	{attribute 'TcIecLibraryType'}
	{attribute 'external_name' := 'F_VN_DrawArrow_GUID_A67F059E_E66C_28C8_6DC9_666EC4C23162'}
	(* Draw an arrowed line. *)
	FUNCTION F_VN_DrawArrow : HRESULT
	VAR_INPUT
		nX1	:	UDINT;	(* x coordinate of the start point *)
		nY1	:	UDINT;	(* y coordinate of the start point *)
		nX2	:	UDINT;	(* x coordinate of the end point *)
		nY2	:	UDINT;	(* y coordinate of the end point *)
		ipDestImage	:	ITcVnImage;	(* Destination image *)
	END_VAR
	VAR_IN_OUT
		aColor	:	TcVnVector4_LREAL;	(* Color *)
	END_VAR
	VAR_INPUT
		nThickness	:	DINT;	(* Line thickness *)
		bDoubleHead	:	BOOL;	(* To draw an arrow on each side of the line. *)
		hrPrev	:	HRESULT;	(* HRESULT indicating the result of previous operations (If SUCCEEDED(hrPrev) equals false, no operation is executed.) *)
	END_VAR

END_FUNCTION

// Functions/Drawing/F_VN_DrawArrow_TcVnVector4_DINT

	{attribute 'TcIecLibraryType'}
	{attribute 'external_name' := 'F_VN_DrawArrow_TcVnVector4_DINT_GUID_4A77EF94_9C2A_22D4_5693_A510294A7600'}
	(* Draw an arrowed line. *)
	FUNCTION F_VN_DrawArrow_TcVnVector4_DINT : HRESULT
	VAR_IN_OUT
		aLine	:	TcVnVector4_DINT;	(* The start and end point of a line segment [x1, y1, x2, y2] *)
	END_VAR
	VAR_INPUT
		ipDestImage	:	ITcVnImage;	(* Destination image *)
	END_VAR
	VAR_IN_OUT
		aColor	:	TcVnVector4_LREAL;	(* Color *)
	END_VAR
	VAR_INPUT
		nThickness	:	DINT;	(* Line thickness *)
		bDoubleHead	:	BOOL;	(* To draw an arrow on each side of the line. *)
		hrPrev	:	HRESULT;	(* HRESULT indicating the result of previous operations (If SUCCEEDED(hrPrev) equals false, no operation is executed.) *)
	END_VAR

END_FUNCTION

// Functions/Drawing/F_VN_DrawArrowExp

	{attribute 'TcIecLibraryType'}
	{attribute 'external_name' := 'F_VN_DrawArrowExp_GUID_1F944010_3B82_22C2_4B5D_AA48D2E539AF'}
	(* Draws an arrowed line. (expert function) *)
	FUNCTION F_VN_DrawArrowExp : HRESULT
	VAR_INPUT
		nX1	:	UDINT;	(* x coordinate of the start point *)
		nY1	:	UDINT;	(* y coordinate of the start point *)
		nX2	:	UDINT;	(* x coordinate of the end point *)
		nY2	:	UDINT;	(* y coordinate of the end point *)
		ipDestImage	:	ITcVnImage;	(* Destination image *)
	END_VAR
	VAR_IN_OUT
		aColor	:	TcVnVector4_LREAL;	(* Color *)
	END_VAR
	VAR_INPUT
		nThickness	:	DINT;	(* Line thickness *)
		bDoubleHead	:	BOOL;	(* To draw an arrow on each side of the line. *)
		eLineType	:	ETcVnLineType;	(* Line type *)
		nShift	:	UDINT;	(* Fractional bits of the coordinates (bit shift) *)
		fTipLenght	:	LREAL;	(* Lenght of the arrow's tip as a fraction of the line's lenght *)
		hrPrev	:	HRESULT;	(* HRESULT indicating the result of previous operations (If SUCCEEDED(hrPrev) equals false, no operation is executed.) *)
	END_VAR

END_FUNCTION

// Functions/Drawing/F_VN_DrawArrowExp_TcVnVector4_DINT

	{attribute 'TcIecLibraryType'}
	{attribute 'external_name' := 'F_VN_DrawArrowExp_TcVnVector4_DINT_GUID_6CFFFCA4_FF10_2C86_53F7_A52292798831'}
	(* Draws an arrowed line. (expert function) *)
	FUNCTION F_VN_DrawArrowExp_TcVnVector4_DINT : HRESULT
	VAR_IN_OUT
		aLine	:	TcVnVector4_DINT;	(* The start and end point of a line segment [x1, y1, x2, y2] *)
	END_VAR
	VAR_INPUT
		ipDestImage	:	ITcVnImage;	(* Destination image *)
	END_VAR
	VAR_IN_OUT
		aColor	:	TcVnVector4_LREAL;	(* Color *)
	END_VAR
	VAR_INPUT
		nThickness	:	DINT;	(* Line thickness *)
		bDoubleHead	:	BOOL;	(* To draw an arrow on each side of the line. *)
		eLineType	:	ETcVnLineType;	(* Line type *)
		nShift	:	UDINT;	(* Fractional bits of the coordinates (bit shift) *)
		fTipLenght	:	LREAL;	(* Lenght of the arrow's tip as a fraction of the line's lenght *)
		hrPrev	:	HRESULT;	(* HRESULT indicating the result of previous operations (If SUCCEEDED(hrPrev) equals false, no operation is executed.) *)
	END_VAR

END_FUNCTION

// Functions/Drawing/F_VN_DrawCircle

	{attribute 'TcIecLibraryType'}
	{attribute 'external_name' := 'F_VN_DrawCircle_GUID_62AE57B7_83F4_253D_652A_20281E468BE3'}
	(* Draws a circle. *)
	FUNCTION F_VN_DrawCircle : HRESULT
	VAR_INPUT
		nCenterX	:	UDINT;	(* x coordinate of the center *)
		nCenterY	:	UDINT;	(* y coordinate of the center *)
		nRadius	:	UDINT;	(* Radius *)
		ipDestImage	:	ITcVnImage;	(* Destination image *)
	END_VAR
	VAR_IN_OUT
		aColor	:	TcVnVector4_LREAL;	(* Color *)
	END_VAR
	VAR_INPUT
		nThickness	:	DINT;	(* Line thickness (if negative, the circle is filled) *)
		hrPrev	:	HRESULT;	(* HRESULT indicating the result of previous operations (If SUCCEEDED(hrPrev) equals false, no operation is executed.) *)
	END_VAR

END_FUNCTION

// Functions/Drawing/F_VN_DrawCircleExp

	{attribute 'TcIecLibraryType'}
	{attribute 'external_name' := 'F_VN_DrawCircleExp_GUID_6C116C34_AD29_2F99_4F7E_E03E108A0E54'}
	(* Draws a circle. *)
	FUNCTION F_VN_DrawCircleExp : HRESULT
	VAR_INPUT
		nCenterX	:	UDINT;	(* x coordinate of the center *)
		nCenterY	:	UDINT;	(* y coordinate of the center *)
		nRadius	:	UDINT;	(* Radius *)
		ipDestImage	:	ITcVnImage;	(* Destination image *)
	END_VAR
	VAR_IN_OUT
		aColor	:	TcVnVector4_LREAL;	(* Color *)
	END_VAR
	VAR_INPUT
		nThickness	:	DINT;	(* Line thickness (if negative, the circle is filled) *)
		eLineType	:	ETcVnLineType;	(* Line type *)
		hrPrev	:	HRESULT;	(* HRESULT indicating the result of previous operations (If SUCCEEDED(hrPrev) equals false, no operation is executed.) *)
	END_VAR

END_FUNCTION

// Functions/Drawing/F_VN_DrawCircles

	{attribute 'TcIecLibraryType'}
	{attribute 'external_name' := 'F_VN_DrawCircles_GUID_940A5C9B_16C1_20B9_6145_00E73CD7E7FA'}
	(* Draws circles. *)
	FUNCTION F_VN_DrawCircles : HRESULT
	VAR_INPUT
		ipCircles	:	ITcVnContainer;	(* Container with circles (ContainerType_Vector_TcVnVector3_REAL; Each container element contains the x coordinate of the circle center [0], the y coordinate of the circle center [1], and the radius [2].) *)
		nCircleIndex	:	DINT;	(* Index of a specific circle to be drawn (if negative, all circles within the container are drawn) *)
		ipDestImage	:	ITcVnImage;	(* Destination image *)
	END_VAR
	VAR_IN_OUT
		aColor	:	TcVnVector4_LREAL;	(* Color *)
	END_VAR
	VAR_INPUT
		nThickness	:	DINT;	(* Line thickness (if negative, the circle is filled) *)
		hrPrev	:	HRESULT;	(* HRESULT indicating the result of previous operations (If SUCCEEDED(hrPrev) equals false, no operation is executed.) *)
	END_VAR

END_FUNCTION

// Functions/Drawing/F_VN_DrawCirclesExp

	{attribute 'TcIecLibraryType'}
	{attribute 'external_name' := 'F_VN_DrawCirclesExp_GUID_C7646B92_088A_23BA_64E0_D477B3D449EC'}
	(* Draws circles. (expert function) *)
	FUNCTION F_VN_DrawCirclesExp : HRESULT
	VAR_INPUT
		ipCircles	:	ITcVnContainer;	(* Container with circles (ContainerType_Vector_TcVnVector3_REAL; Each container element contains the x coordinate of the circle center [0], the y coordinate of the circle center [1], and the radius [2].) *)
		nCircleIndex	:	DINT;	(* Index of a specific circle to be drawn (if negative, all circles within the container are drawn) *)
		ipDestImage	:	ITcVnImage;	(* Destination image *)
	END_VAR
	VAR_IN_OUT
		aColor	:	TcVnVector4_LREAL;	(* Color *)
	END_VAR
	VAR_INPUT
		nThickness	:	DINT;	(* Line thickness (if negative, the circle is filled) *)
		eLineType	:	ETcVnLineType;	(* Line type *)
		hrPrev	:	HRESULT;	(* HRESULT indicating the result of previous operations (If SUCCEEDED(hrPrev) equals false, no operation is executed.) *)
	END_VAR

END_FUNCTION

// Functions/Drawing/F_VN_DrawCircularArc

	{attribute 'TcIecLibraryType'}
	{attribute 'external_name' := 'F_VN_DrawCircularArc_GUID_65BA9826_3505_21EA_7421_EA736909BE51'}
	(* Draws a circular arc. *)
	FUNCTION F_VN_DrawCircularArc : HRESULT
	VAR_IN_OUT
		stCircularArc	:	TcVnCircularArc;	(* Circular arc definition *)
	END_VAR
	VAR_INPUT
		ipDestImage	:	ITcVnImage;	(* Destination image *)
	END_VAR
	VAR_IN_OUT
		aColor	:	TcVnVector4_LREAL;	(* Color *)
	END_VAR
	VAR_INPUT
		nThickness	:	DINT;	(* Line thickness (if negative, the arc is filled) *)
		hrPrev	:	HRESULT;	(* HRESULT indicating the result of previous operations (If SUCCEEDED(hrPrev) equals false, no operation is executed.) *)
	END_VAR

END_FUNCTION

// Functions/Drawing/F_VN_DrawCircularArcExp

	{attribute 'TcIecLibraryType'}
	{attribute 'external_name' := 'F_VN_DrawCircularArcExp_GUID_5E53D375_1C4A_2CA0_6893_A6AF5257BA9F'}
	(* Draws a circular arc. (expert function) *)
	FUNCTION F_VN_DrawCircularArcExp : HRESULT
	VAR_IN_OUT
		stCircularArc	:	TcVnCircularArc;	(* Circular arc definition *)
	END_VAR
	VAR_INPUT
		ipDestImage	:	ITcVnImage;	(* Destination image *)
	END_VAR
	VAR_IN_OUT
		aColor	:	TcVnVector4_LREAL;	(* Color *)
	END_VAR
	VAR_INPUT
		nThickness	:	DINT;	(* Line thickness (if negative, the arc is filled) *)
		eLineType	:	ETcVnLineType;	(* Line type *)
		hrPrev	:	HRESULT;	(* HRESULT indicating the result of previous operations (If SUCCEEDED(hrPrev) equals false, no operation is executed.) *)
	END_VAR

END_FUNCTION

// Functions/Drawing/F_VN_DrawComponents

	{attribute 'TcIecLibraryType'}
	{attribute 'external_name' := 'F_VN_DrawComponents_GUID_6E728B5E_19B3_2D00_71CC_5B002C0B6E3E'}
	(* Draw the results of connected component function. *)
	FUNCTION F_VN_DrawComponents : HRESULT
	VAR_INPUT
		ipLabelImage	:	ITcVnImage;	(* Image contains labels for each pixel (1 channel DINT or UINT). *)
		nLabelID	:	DINT;	(* Value of a specific label to be drawn (if negative, all components within the image are drawn) *)
		ipDestImage	:	REFERENCE TO ITcVnImage;	(* Destination image (An appropriate image will be created if required. The output image is 1 or 3 channels USINT). *)
		bShowLabelID	:	BOOL;	(* Show label ID in the center of the component on the destination image *)
		hrPrev	:	HRESULT;	(* HRESULT indicating the result of previous operations (If SUCCEEDED(hrPrev) equals false, no operation is executed.) *)
	END_VAR

END_FUNCTION

// Functions/Drawing/F_VN_DrawComponentsExp

	{attribute 'TcIecLibraryType'}
	{attribute 'external_name' := 'F_VN_DrawComponentsExp_GUID_E0170EF0_CACF_258E_7E4E_5469F394004B'}
	(* Draw the results of connected component function. (expert function) *)
	FUNCTION F_VN_DrawComponentsExp : HRESULT
	VAR_INPUT
		ipLabelImage	:	ITcVnImage;	(* Image contains labels for each pixel (1 channel DINT or UINT). *)
		nLabelID	:	DINT;	(* Value of a specific label to be drawn (if negative, all components within the image are drawn) *)
		ipDestImage	:	REFERENCE TO ITcVnImage;	(* Destination image (An appropriate image will be created if required. The output image is 1 or 3 channels USINT). *)
		bShowLabelID	:	BOOL;	(* Show lable ID in the center of the component on the destination image *)
	END_VAR
	VAR_IN_OUT
		aColor	:	TcVnVector4_LREAL;	(* Color to draw the components (for {-1, -1, -1, -1}, a random color is chosen for each component) *)
	END_VAR
	VAR_INPUT
		nThickness	:	DINT;	(* Text line thickness *)
		fFontScale	:	LREAL;	(* Scaling factor for the text *)
		hrPrev	:	HRESULT;	(* HRESULT indicating the result of previous operations (If SUCCEEDED(hrPrev) equals false, no operation is executed.) *)
	END_VAR

END_FUNCTION

// Functions/Drawing/F_VN_DrawContours

	{attribute 'TcIecLibraryType'}
	{attribute 'external_name' := 'F_VN_DrawContours_GUID_3A760F26_AE23_21F0_7549_3A204CDE6949'}
	(* Draws a single point set or multiple point sets that are interpreted as contours. *)
	FUNCTION F_VN_DrawContours : HRESULT
	VAR_INPUT
		ipContours	:	ITcVnContainer;	(* Single contour (ContainerType_Vector_TcVnPoint2_DINT) or multiple contours (ContainerType_Vector_Vector_TcVnPoint2_DINT) *)
		nContourIndex	:	DINT;	(* Index of a specific contour to be drawn (if negative, all contours within the container are drawn) *)
		ipDestImage	:	ITcVnImage;	(* Destination image *)
	END_VAR
	VAR_IN_OUT
		aColor	:	TcVnVector4_LREAL;	(* Color *)
	END_VAR
	VAR_INPUT
		nThickness	:	DINT;	(* Line thickness (if negative, the contours are filled) *)
		hrPrev	:	HRESULT;	(* HRESULT indicating the result of previous operations (If SUCCEEDED(hrPrev) equals false, no operation is executed.) *)
	END_VAR

END_FUNCTION

// Functions/Drawing/F_VN_DrawContoursExp

	{attribute 'TcIecLibraryType'}
	{attribute 'external_name' := 'F_VN_DrawContoursExp_GUID_491B5FE3_1D62_2512_69DC_BD3D74F64591'}
	(* Draws a single point set or multiple point sets that are interpreted as contours. (expert function) *)
	FUNCTION F_VN_DrawContoursExp : HRESULT
	VAR_INPUT
		ipContours	:	ITcVnContainer;	(* Single contour (ContainerType_Vector_TcVnPoint2_DINT) or multiple contours (ContainerType_Vector_Vector_TcVnPoint2_DINT) *)
		nContourIndex	:	DINT;	(* Index of a specific contour to be drawn (if negative, all contours within the container are drawn) *)
		ipDestImage	:	ITcVnImage;	(* Destination image *)
	END_VAR
	VAR_IN_OUT
		aColor	:	TcVnVector4_LREAL;	(* Color *)
	END_VAR
	VAR_INPUT
		nThickness	:	DINT;	(* Line thickness (if negative, the contours are filled) *)
		eLineType	:	ETcVnLineType;	(* Line type *)
		ipHierarchy	:	ITcVnContainer;	(* Contour hierarchy (ContainerType_Vector_TcVnVector4_DINT) *)
		nMaxLevel	:	DINT;	(* Maximum level of contours to be drawn *)
	END_VAR
	VAR_IN_OUT
		aOffset	:	TcVnPoint;	(* Offset by which every contour point is shifted *)
	END_VAR
	VAR_INPUT
		hrPrev	:	HRESULT;	(* HRESULT indicating the result of previous operations (If SUCCEEDED(hrPrev) equals false, no operation is executed.) *)
	END_VAR

END_FUNCTION

// Functions/Drawing/F_VN_DrawEllipse

	{attribute 'TcIecLibraryType'}
	{attribute 'external_name' := 'F_VN_DrawEllipse_GUID_B36BA161_2BCF_2E35_626D_D9A20308391B'}
	(* Draws an ellipse. *)
	FUNCTION F_VN_DrawEllipse : HRESULT
	VAR_IN_OUT
		stEllipse	:	TcVnRotatedRectangle;	(* Ellipse to be drawn (rotation angle in degrees) *)
	END_VAR
	VAR_INPUT
		ipDestImage	:	ITcVnImage;	(* Destination image *)
	END_VAR
	VAR_IN_OUT
		aColor	:	TcVnVector4_LREAL;	(* Color *)
	END_VAR
	VAR_INPUT
		nThickness	:	DINT;	(* Line thickness (if negative, the ellipse is filled) *)
		hrPrev	:	HRESULT;	(* HRESULT indicating the result of previous operations (If SUCCEEDED(hrPrev) equals false, no operation is executed.) *)
	END_VAR

END_FUNCTION

// Functions/Drawing/F_VN_DrawEllipseExp

	{attribute 'TcIecLibraryType'}
	{attribute 'external_name' := 'F_VN_DrawEllipseExp_GUID_4267312D_E9F9_285D_445A_87EE5A0952CB'}
	(* Draws an ellipse. (expert function) *)
	FUNCTION F_VN_DrawEllipseExp : HRESULT
	VAR_IN_OUT
		stEllipse	:	TcVnRotatedRectangle;	(* Ellipse to be drawn (rotation angle in degrees) *)
	END_VAR
	VAR_INPUT
		ipDestImage	:	ITcVnImage;	(* Destination image *)
	END_VAR
	VAR_IN_OUT
		aColor	:	TcVnVector4_LREAL;	(* Color *)
	END_VAR
	VAR_INPUT
		nThickness	:	DINT;	(* Line thickness (if negative, the ellipse is filled) *)
		eLineType	:	ETcVnLineType;	(* Line type *)
		hrPrev	:	HRESULT;	(* HRESULT indicating the result of previous operations (If SUCCEEDED(hrPrev) equals false, no operation is executed.) *)
	END_VAR

END_FUNCTION

// Functions/Drawing/F_VN_DrawKeypoints

	{attribute 'TcIecLibraryType'}
	{attribute 'external_name' := 'F_VN_DrawKeypoints_GUID_FB38EC14_E7EA_2A28_6ADF_7A92046F99E5'}
	(* Draws the keypoints for visualization purpose. *)
	FUNCTION F_VN_DrawKeypoints : HRESULT
	VAR_INPUT
		ipSrcImage	:	ITcVnImage;	(* Source image (elements of type USINT) *)
		ipKeyPoints	:	ITcVnContainer;	(* Container with the keypoints (ContainerType_Vector_TcVnKeyPoint) *)
		ipDestImage	:	REFERENCE TO ITcVnImage;	(* Destination image (An appropriate color image will be created if required.) *)
		hrPrev	:	HRESULT;	(* HRESULT indicating the result of previous operations (If SUCCEEDED(hrPrev) equals false, no operation is executed.) *)
	END_VAR

END_FUNCTION

// Functions/Drawing/F_VN_DrawKeypointsExp

	{attribute 'TcIecLibraryType'}
	{attribute 'external_name' := 'F_VN_DrawKeypointsExp_GUID_5513617A_5140_2AEB_572F_A22AF2CF3272'}
	(* Draws the keypoints for visualization purpose. (expert function) *)
	FUNCTION F_VN_DrawKeypointsExp : HRESULT
	VAR_INPUT
		ipSrcImage	:	ITcVnImage;	(* Source image (elements of type USINT) *)
		ipKeyPoints	:	ITcVnContainer;	(* Container with the keypoints (ContainerType_Vector_TcVnKeyPoint) *)
		ipDestImage	:	REFERENCE TO ITcVnImage;	(* Destination image (An appropriate color image will be created if required.) *)
	END_VAR
	VAR_IN_OUT
		aColor	:	TcVnVector4_LREAL;	(* Color to draw the keypoints (for {-1, -1, -1, -1}, a random color is chosen for each point) *)
	END_VAR
	VAR_INPUT
		eFlags	:	ETcVnDrawMatchesFlags;	(* A combination of flags to support overdrawing an existing destination image and/or drawing additional (Rich-)Keypoint information (size and orientation) *)
		hrPrev	:	HRESULT;	(* HRESULT indicating the result of previous operations (If SUCCEEDED(hrPrev) equals false, no operation is executed.) *)
	END_VAR

END_FUNCTION

// Functions/Drawing/F_VN_DrawLine

	{attribute 'TcIecLibraryType'}
	{attribute 'external_name' := 'F_VN_DrawLine_GUID_859089CD_2CB1_20E2_51BC_E78BFF23C3ED'}
	(* Draws a line. *)
	FUNCTION F_VN_DrawLine : HRESULT
	VAR_INPUT
		nX1	:	UDINT;	(* x coordinate of the start point *)
		nY1	:	UDINT;	(* y coordinate of the start point *)
		nX2	:	UDINT;	(* x coordinate of the end point *)
		nY2	:	UDINT;	(* y coordinate of the end point *)
		ipDestImage	:	ITcVnImage;	(* Destination image *)
	END_VAR
	VAR_IN_OUT
		aColor	:	TcVnVector4_LREAL;	(* Color *)
	END_VAR
	VAR_INPUT
		nThickness	:	DINT;	(* Line thickness *)
		hrPrev	:	HRESULT;	(* HRESULT indicating the result of previous operations (If SUCCEEDED(hrPrev) equals false, no operation is executed.) *)
	END_VAR

END_FUNCTION

// Functions/Drawing/F_VN_DrawLineExp

	{attribute 'TcIecLibraryType'}
	{attribute 'external_name' := 'F_VN_DrawLineExp_GUID_DDC0CE2F_05D8_23C1_7C2F_F01A04BF4976'}
	(* Draws a line. (expert function) *)
	FUNCTION F_VN_DrawLineExp : HRESULT
	VAR_INPUT
		nX1	:	UDINT;	(* x coordinate of the start point *)
		nY1	:	UDINT;	(* y coordinate of the start point *)
		nX2	:	UDINT;	(* x coordinate of the end point *)
		nY2	:	UDINT;	(* y coordinate of the end point *)
		ipDestImage	:	ITcVnImage;	(* Destination image *)
	END_VAR
	VAR_IN_OUT
		aColor	:	TcVnVector4_LREAL;	(* Color *)
	END_VAR
	VAR_INPUT
		nThickness	:	DINT;	(* Line thickness *)
		eLineType	:	ETcVnLineType;	(* Line type *)
		nShift	:	UDINT;	(* Fractional bits of the coordinates (bit shift) *)
		hrPrev	:	HRESULT;	(* HRESULT indicating the result of previous operations (If SUCCEEDED(hrPrev) equals false, no operation is executed.) *)
	END_VAR

END_FUNCTION

// Functions/Drawing/F_VN_DrawLine_TcVnVector4_DINT

	{attribute 'TcIecLibraryType'}
	{attribute 'external_name' := 'F_VN_DrawLine_TcVnVector4_DINT_GUID_0BCA7416_8C02_23F6_5098_9813FC3D218D'}
	(* Draws a line. *)
	FUNCTION F_VN_DrawLine_TcVnVector4_DINT : HRESULT
	VAR_IN_OUT
		aLine	:	TcVnVector4_DINT;	(* The start and end point of a line segment [x1, y1, x2, y2] *)
	END_VAR
	VAR_INPUT
		ipDestImage	:	ITcVnImage;	(* Destination image *)
	END_VAR
	VAR_IN_OUT
		aColor	:	TcVnVector4_LREAL;	(* Color *)
	END_VAR
	VAR_INPUT
		nThickness	:	DINT;	(* Line thickness *)
		hrPrev	:	HRESULT;	(* HRESULT indicating the result of previous operations (If SUCCEEDED(hrPrev) equals false, no operation is executed.) *)
	END_VAR

END_FUNCTION

// Functions/Drawing/F_VN_DrawLineExp_TcVnVector4_DINT

	{attribute 'TcIecLibraryType'}
	{attribute 'external_name' := 'F_VN_DrawLineExp_TcVnVector4_DINT_GUID_6BA4293A_6958_2BBA_5CA1_9439207B768B'}
	(* Draws a line. (expert function) *)
	FUNCTION F_VN_DrawLineExp_TcVnVector4_DINT : HRESULT
	VAR_IN_OUT
		aLine	:	TcVnVector4_DINT;	(* The start and end point of a line segment [x1, y1, x2, y2] *)
	END_VAR
	VAR_INPUT
		ipDestImage	:	ITcVnImage;	(* Destination image *)
	END_VAR
	VAR_IN_OUT
		aColor	:	TcVnVector4_LREAL;	(* Color *)
	END_VAR
	VAR_INPUT
		nThickness	:	DINT;	(* Line thickness *)
		eLineType	:	ETcVnLineType;	(* Line type *)
		nShift	:	UDINT;	(* Fractional bits of the coordinates (bit shift) *)
		hrPrev	:	HRESULT;	(* HRESULT indicating the result of previous operations (If SUCCEEDED(hrPrev) equals false, no operation is executed.) *)
	END_VAR

END_FUNCTION

// Functions/Drawing/F_VN_DrawLine_TcVnVector4_LREAL

	{attribute 'TcIecLibraryType'}
	{attribute 'external_name' := 'F_VN_DrawLine_TcVnVector4_LREAL_GUID_F0143CEA_0B4A_2A30_6B90_6C5F1AF27D68'}
	(* Draws a line. *)
	FUNCTION F_VN_DrawLine_TcVnVector4_LREAL : HRESULT
	VAR_IN_OUT
		aLine	:	TcVnVector4_LREAL;	(* The first and second element describe the x and y component of the direction vector. The third and fourth element describe the x and y component of the position vector. *)
	END_VAR
	VAR_INPUT
		ipDestImage	:	ITcVnImage;	(* Destination image *)
	END_VAR
	VAR_IN_OUT
		aColor	:	TcVnVector4_LREAL;	(* Color *)
	END_VAR
	VAR_INPUT
		nThickness	:	DINT;	(* Line thickness *)
		hrPrev	:	HRESULT;	(* HRESULT indicating the result of previous operations (If SUCCEEDED(hrPrev) equals false, no operation is executed.) *)
	END_VAR

END_FUNCTION

// Functions/Drawing/F_VN_DrawLineExp_TcVnVector4_LREAL

	{attribute 'TcIecLibraryType'}
	{attribute 'external_name' := 'F_VN_DrawLineExp_TcVnVector4_LREAL_GUID_497D2B2B_F8A5_2B06_68D9_A8BDD2C62665'}
	(* Draws a line. (expert function) *)
	FUNCTION F_VN_DrawLineExp_TcVnVector4_LREAL : HRESULT
	VAR_IN_OUT
		aLine	:	TcVnVector4_LREAL;	(* The first and second element describe the x and y component of the direction vector. The third and fourth element describe the x and y component of the position vector. *)
	END_VAR
	VAR_INPUT
		ipDestImage	:	ITcVnImage;	(* Destination image *)
	END_VAR
	VAR_IN_OUT
		aColor	:	TcVnVector4_LREAL;	(* Color *)
	END_VAR
	VAR_INPUT
		nThickness	:	DINT;	(* Line thickness *)
		eLineType	:	ETcVnLineType;	(* Line type *)
		nShift	:	UDINT;	(* Fractional bits of the coordinates (bit shift) *)
		hrPrev	:	HRESULT;	(* HRESULT indicating the result of previous operations (If SUCCEEDED(hrPrev) equals false, no operation is executed.) *)
	END_VAR

END_FUNCTION

// Functions/Drawing/F_VN_DrawLines

	{attribute 'TcIecLibraryType'}
	{attribute 'external_name' := 'F_VN_DrawLines_GUID_7FF7FF3E_D555_2BC9_6EE9_83C9F1D24540'}
	(* Draws lines. *)
	FUNCTION F_VN_DrawLines : HRESULT
	VAR_INPUT
		ipLines	:	ITcVnContainer;	(* Container with line descriptions (ContainerType_Vector_TcVnVector2_REAL: the distance from the origin [0] in pixels and the rotation angle [1] in radians. ContainerType_Vector_TcVnVector4_LREAL: the first and second element describe the x and y component of a vector collinear to the line. The third and fourth element describe the x and y component of a point on the line. ContainerType_Vector_TcVnVector4_DINT: start and end point [x1, y1, x2, y2]) *)
		nLineIndex	:	DINT;	(* Index of a specific line to be drawn (if negative, all lines within the container are drawn) *)
		ipDestImage	:	ITcVnImage;	(* Destination image *)
	END_VAR
	VAR_IN_OUT
		aColor	:	TcVnVector4_LREAL;	(* Color *)
	END_VAR
	VAR_INPUT
		nThickness	:	DINT;	(* Line thickness *)
		hrPrev	:	HRESULT;	(* HRESULT indicating the result of previous operations (If SUCCEEDED(hrPrev) equals false, no operation is executed.) *)
	END_VAR

END_FUNCTION

// Functions/Drawing/F_VN_DrawLinesExp

	{attribute 'TcIecLibraryType'}
	{attribute 'external_name' := 'F_VN_DrawLinesExp_GUID_44E45FE5_8AEB_2A9E_7E98_0C10B83BCE72'}
	(* Draws lines. (expert function) *)
	FUNCTION F_VN_DrawLinesExp : HRESULT
	VAR_INPUT
		ipLines	:	ITcVnContainer;	(* Container with line descriptions (ContainerType_Vector_TcVnVector2_REAL: the distance from the origin [0] in pixels and the rotation angle [1] in radians. ContainerType_Vector_TcVnVector4_LREAL: the first and second element describe the x and y component of a vector collinear to the line. The third and fourth element describe the x and y component of a point on the line. ContainerType_Vector_TcVnVector4_DINT: start and end point [x1, y1, x2, y2]) *)
		nLineIndex	:	DINT;	(* Index of a specific line to be drawn (if negative, all lines within the container are drawn) *)
		ipDestImage	:	ITcVnImage;	(* Destination image *)
	END_VAR
	VAR_IN_OUT
		aColor	:	TcVnVector4_LREAL;	(* Color *)
	END_VAR
	VAR_INPUT
		nThickness	:	DINT;	(* Line thickness *)
		eLineType	:	ETcVnLineType;	(* Line type *)
		nShift	:	UDINT;	(* Fractional bits of the coordinates (bit shift) *)
		hrPrev	:	HRESULT;	(* HRESULT indicating the result of previous operations (If SUCCEEDED(hrPrev) equals false, no operation is executed.) *)
	END_VAR

END_FUNCTION

// Functions/Drawing/F_VN_DrawMatches

	{attribute 'TcIecLibraryType'}
	{attribute 'external_name' := 'F_VN_DrawMatches_GUID_942AD279_6BB1_2A54_440D_B19BA420E0BA'}
	(* Draws the keypoints and matches for visualization purpose. *)
	FUNCTION F_VN_DrawMatches : HRESULT
	VAR_INPUT
		ipSrcImage1	:	ITcVnImage;	(* Source image 1 (elements of type USINT) *)
		ipKeyPoints1	:	ITcVnContainer;	(* Container with the keypoints 1 (ContainerType_Vector_TcVnKeyPoint) *)
		ipSrcImage2	:	ITcVnImage;	(* Source image 2 (elements of type USINT, must have the same number of channels as ipSrcImage1) *)
		ipKeyPoints2	:	ITcVnContainer;	(* Container with the keypoints 2 (ContainerType_Vector_TcVnKeyPoint) *)
		ipMatches1To2	:	ITcVnContainer;	(* Container with the descriptor matches (ContainerType_Vector_TcVnDMatch) *)
		ipDestImage	:	REFERENCE TO ITcVnImage;	(* Destination image (An appropriate color image will be created if required.) *)
		hrPrev	:	HRESULT;	(* HRESULT indicating the result of previous operations (If SUCCEEDED(hrPrev) equals false, no operation is executed.) *)
	END_VAR

END_FUNCTION

// Functions/Drawing/F_VN_DrawMatchesExp

	{attribute 'TcIecLibraryType'}
	{attribute 'external_name' := 'F_VN_DrawMatchesExp_GUID_DE93B311_EDEA_2A84_5CE6_E45424376C21'}
	(* Draws the keypoints and matches for visualization purpose. (expert function) *)
	FUNCTION F_VN_DrawMatchesExp : HRESULT
	VAR_INPUT
		ipSrcImage1	:	ITcVnImage;	(* Source image 1 (elements of type USINT) *)
		ipKeyPoints1	:	ITcVnContainer;	(* Container with the keypoints 1 (ContainerType_Vector_TcVnKeyPoint) *)
		ipSrcImage2	:	ITcVnImage;	(* Source image 2 (elements of type USINT, must have the same number of channels as ipSrcImage1) *)
		ipKeyPoints2	:	ITcVnContainer;	(* Container with the keypoints 2 (ContainerType_Vector_TcVnKeyPoint) *)
		ipMatches1To2	:	ITcVnContainer;	(* Container with the descriptor matches (ContainerType_Vector_TcVnDMatch) *)
		ipDestImage	:	REFERENCE TO ITcVnImage;	(* Destination image (An appropriate color image will be created if required.) *)
	END_VAR
	VAR_IN_OUT
		aMatchColor	:	TcVnVector4_LREAL;	(* Color to draw the matches (for {-1, -1, -1, -1}, a random color is chosen for each point and line) *)
		aSingleColor	:	TcVnVector4_LREAL;	(* Color to draw the single keypoints (for {-1, -1, -1, -1}, a random color is chosen for each point) *)
	END_VAR
	VAR_INPUT
		ipMatchesMask	:	ITcVnContainer;	(* Mask to select the matches to be drawn (ContainerType_Vector_SINT; Set to 0 if all matches should be drawn.) *)
		eFlags	:	ETcVnDrawMatchesFlags;	(* A combination of flags to support overdrawing an existing destination image and/or drawing additional (Rich-)Keypoint information (size and orientation) and/or skipping single keypoints *)
		hrPrev	:	HRESULT;	(* HRESULT indicating the result of previous operations (If SUCCEEDED(hrPrev) equals false, no operation is executed.) *)
	END_VAR

END_FUNCTION

// Functions/Drawing/F_VN_DrawOrientation

	{attribute 'TcIecLibraryType'}
	{attribute 'external_name' := 'F_VN_DrawOrientation_GUID_945177D4_9B20_2F7A_5F29_B2DEFC5FDA37'}
	(* Draw the main axis of a set of points/contour based on a rotated rectangle. *)
	FUNCTION F_VN_DrawOrientation : HRESULT
	VAR_IN_OUT
		stOrientation	:	TcVnRotatedRectangle;	(* Rotated rectangle, containig center of mass, lenghts of axes, and rotation angle in clockwise direction *)
	END_VAR
	VAR_INPUT
		ipDestImage	:	ITcVnImage;	(* Destination image *)
	END_VAR
	VAR_IN_OUT
		aColorMainAxis	:	TcVnVector4_LREAL;	(* Color of the major axis *)
	END_VAR
	VAR_INPUT
		nThickness	:	DINT;	(* Line thickness *)
		hrPrev	:	HRESULT;	(* HRESULT indicating the result of previous operations (If SUCCEEDED(hrPrev) equals false, no operation is executed.) *)
	END_VAR

END_FUNCTION

// Functions/Drawing/F_VN_DrawOrientationExp

	{attribute 'TcIecLibraryType'}
	{attribute 'external_name' := 'F_VN_DrawOrientationExp_GUID_71610F20_995C_2595_6B24_5DB885A560D9'}
	(* Draw the main axis, the horizontal axis and the angle of a set of points/contour based on a rotated rectangle. (expert function) *)
	FUNCTION F_VN_DrawOrientationExp : HRESULT
	VAR_IN_OUT
		stOrientation	:	TcVnRotatedRectangle;	(* Rotated rectangle, containig center of mass, lenghts of axes, and rotation angle in clockwise direction *)
	END_VAR
	VAR_INPUT
		ipDestImage	:	ITcVnImage;	(* Destination image *)
	END_VAR
	VAR_IN_OUT
		aColorMainAxis	:	TcVnVector4_LREAL;	(* Color of the major axis *)
	END_VAR
	VAR_INPUT
		nThickness	:	DINT;	(* Line thickness *)
	END_VAR
	VAR_IN_OUT
		aColorHorizontalAxis	:	TcVnVector4_LREAL;	(* Color of the horizontal axis *)
	END_VAR
	VAR_INPUT
		fFontScale	:	LREAL;	(* Scaling factor for the text *)
		hrPrev	:	HRESULT;	(* HRESULT indicating the result of previous operations (If SUCCEEDED(hrPrev) equals false, no operation is executed.) *)
	END_VAR

END_FUNCTION

// Functions/Drawing/F_VN_DrawPoint

	{attribute 'TcIecLibraryType'}
	{attribute 'external_name' := 'F_VN_DrawPoint_GUID_F314C2B7_1A60_2C17_7ED9_866531D08079'}
	(* Draws a point. *)
	FUNCTION F_VN_DrawPoint : HRESULT
	VAR_INPUT
		nX	:	UDINT;	(* x coordinate of the point *)
		nY	:	UDINT;	(* y coordinate of the point *)
		ipDestImage	:	ITcVnImage;	(* Destination image *)
		eShape	:	ETcVnDrawShape;	(* Point shape *)
	END_VAR
	VAR_IN_OUT
		aColor	:	TcVnVector4_LREAL;	(* Color (for {-1, -1, -1, -1}, a random color is chosen) *)
	END_VAR
	VAR_INPUT
		hrPrev	:	HRESULT;	(* HRESULT indicating the result of previous operations (If SUCCEEDED(hrPrev) equals false, no operation is executed.) *)
	END_VAR

END_FUNCTION

// Functions/Drawing/F_VN_DrawPointExp

	{attribute 'TcIecLibraryType'}
	{attribute 'external_name' := 'F_VN_DrawPointExp_GUID_14BC56EB_7489_25AD_41C6_BE616B054DCA'}
	(* Draw a point. (expert function) *)
	FUNCTION F_VN_DrawPointExp : HRESULT
	VAR_INPUT
		nX	:	UDINT;	(* x coordinate of the point *)
		nY	:	UDINT;	(* y coordinate of the point *)
		ipDestImage	:	ITcVnImage;	(* Destination image *)
		eShape	:	ETcVnDrawShape;	(* Point shape *)
	END_VAR
	VAR_IN_OUT
		aColor	:	TcVnVector4_LREAL;	(* Color (for {-1, -1, -1, -1}, a random color is chosen) *)
	END_VAR
	VAR_INPUT
		nSize	:	UDINT;	(* Size of the shape (half width) *)
		nThickness	:	DINT;	(* Line thickness (if negative, the shape is filled if it is closed) *)
		eLineType	:	ETcVnLineType;	(* Line type *)
		hrPrev	:	HRESULT;	(* HRESULT indicating the result of previous operations (If SUCCEEDED(hrPrev) equals false, no operation is executed.) *)
	END_VAR

END_FUNCTION

// Functions/Drawing/F_VN_DrawPoints

	{attribute 'TcIecLibraryType'}
	{attribute 'external_name' := 'F_VN_DrawPoints_GUID_FEC580F2_7856_254F_576C_68C6A0E88178'}
	(* Draw a collection of points. *)
	FUNCTION F_VN_DrawPoints : HRESULT
	VAR_INPUT
		ipPoints	:	ITcVnContainer;	(* Container with TcVnPoint2_DINT or TcVnPoint2_REAL elements *)
		ipDestImage	:	ITcVnImage;	(* Destination image *)
		eShape	:	ETcVnDrawShape;	(* Point shape *)
	END_VAR
	VAR_IN_OUT
		aColor	:	TcVnVector4_LREAL;	(* Color (for {-1, -1, -1, -1}, a random color is chosen for each point) *)
	END_VAR
	VAR_INPUT
		hrPrev	:	HRESULT;	(* HRESULT indicating the result of previous operations (If SUCCEEDED(hrPrev) equals false, no operation is executed.) *)
	END_VAR

END_FUNCTION

// Functions/Drawing/F_VN_DrawPointsExp

	{attribute 'TcIecLibraryType'}
	{attribute 'external_name' := 'F_VN_DrawPointsExp_GUID_2CBF2F26_77DD_2731_479E_892A60F2DFB1'}
	(* Draw a collection of points. (expert function) *)
	FUNCTION F_VN_DrawPointsExp : HRESULT
	VAR_INPUT
		ipPoints	:	ITcVnContainer;	(* Container with TcVnPoint2_DINT or TcVnPoint2_REAL elements *)
		ipDestImage	:	ITcVnImage;	(* Destination image *)
		eShape	:	ETcVnDrawShape;	(* Point shape *)
	END_VAR
	VAR_IN_OUT
		aColor	:	TcVnVector4_LREAL;	(* Color (for {-1, -1, -1, -1}, a random color is chosen for each point) *)
	END_VAR
	VAR_INPUT
		nSize	:	UDINT;	(* Size of the shape (half width) *)
		nThickness	:	DINT;	(* Line thickness (if negative, the shape is filled if it is closed) *)
		eLineType	:	ETcVnLineType;	(* Line type *)
		hrPrev	:	HRESULT;	(* HRESULT indicating the result of previous operations (If SUCCEEDED(hrPrev) equals false, no operation is executed.) *)
	END_VAR

END_FUNCTION

// Functions/Drawing/F_VN_DrawPolygon

	{attribute 'TcIecLibraryType'}
	{attribute 'external_name' := 'F_VN_DrawPolygon_GUID_32CE6F2D_7A8C_26C8_4266_5FCEBE7E61DF'}
	(* Draw a pologon using collection of points. *)
	FUNCTION F_VN_DrawPolygon : HRESULT
	VAR_INPUT
		ipPoints	:	ITcVnContainer;	(* Container with TcVnPoint2_DINT, TcVnPoint2_REAL, or TcVnPoint2_LREAL elements *)
		ipDestImage	:	ITcVnImage;	(* Destination image *)
	END_VAR
	VAR_IN_OUT
		aColor	:	TcVnVector4_LREAL;	(* Color *)
	END_VAR
	VAR_INPUT
		nThickness	:	DINT;	(* Line thickness (if negative, the polygon is filled) *)
		hrPrev	:	HRESULT;	(* HRESULT indicating the result of previous operations (If SUCCEEDED(hrPrev) equals false, no operation is executed.) *)
	END_VAR

END_FUNCTION

// Functions/Drawing/F_VN_DrawPolygonExp

	{attribute 'TcIecLibraryType'}
	{attribute 'external_name' := 'F_VN_DrawPolygonExp_GUID_CF972D1A_F834_2AC1_4D96_1C0649D86EAA'}
	(* Draw a pologon using collection of points. (expert function) *)
	FUNCTION F_VN_DrawPolygonExp : HRESULT
	VAR_INPUT
		ipPoints	:	ITcVnContainer;	(* Container with TcVnPoint2_DINT, TcVnPoint2_REAL, or TcVnPoint2_LREAL elements *)
		ipDestImage	:	ITcVnImage;	(* Destination image *)
	END_VAR
	VAR_IN_OUT
		aColor	:	TcVnVector4_LREAL;	(* Color *)
	END_VAR
	VAR_INPUT
		nThickness	:	DINT;	(* Line thickness (if negative, the shape is filled) *)
		bIsClosed	:	BOOL;	(* If it is true, the function draws a line from the last point to the first point to close the polygon. *)
		eLineType	:	ETcVnLineType;	(* Line type *)
		nShift	:	UDINT;	(* Fractional bits of the coordinates (bit shift) *)
		hrPrev	:	HRESULT;	(* HRESULT indicating the result of previous operations (If SUCCEEDED(hrPrev) equals false, no operation is executed.) *)
	END_VAR

END_FUNCTION

// Functions/Drawing/F_VN_DrawRectangle

	{attribute 'TcIecLibraryType'}
	{attribute 'external_name' := 'F_VN_DrawRectangle_GUID_D27B98D0_3450_254A_5B1B_E2030FE9D66E'}
	(* Draw a rectangle. *)
	FUNCTION F_VN_DrawRectangle : HRESULT
	VAR_INPUT
		nTopLeftX	:	UDINT;	(* x coordinate of the top left corner *)
		nTopLeftY	:	UDINT;	(* y coordinate of the top left corner *)
		nBottomRightX	:	UDINT;	(* x coordinate of the bottom right corner *)
		nBottomRightY	:	UDINT;	(* y coordinate of the bottom right corner *)
		ipDestImage	:	ITcVnImage;	(* Destination image *)
	END_VAR
	VAR_IN_OUT
		aColor	:	TcVnVector4_LREAL;	(* Color *)
	END_VAR
	VAR_INPUT
		nThickness	:	DINT;	(* Line thickness (if negative, the rectangle is filled) *)
		hrPrev	:	HRESULT;	(* HRESULT indicating the result of previous operations (If SUCCEEDED(hrPrev) equals false, no operation is executed.) *)
	END_VAR

END_FUNCTION

// Functions/Drawing/F_VN_DrawRectangle_TcVnRectangle_DINT

	{attribute 'TcIecLibraryType'}
	{attribute 'external_name' := 'F_VN_DrawRectangle_TcVnRectangle_DINT_GUID_2D98B81A_DC59_2558_61FD_E38D454CD2B7'}
	(* Draw a rectangle. *)
	FUNCTION F_VN_DrawRectangle_TcVnRectangle_DINT : HRESULT
	VAR_IN_OUT
		stRectangle	:	TcVnRectangle_DINT;	(* Rectangle to be drawn *)
	END_VAR
	VAR_INPUT
		ipDestImage	:	ITcVnImage;	(* Destination image *)
	END_VAR
	VAR_IN_OUT
		aColor	:	TcVnVector4_LREAL;	(* Color *)
	END_VAR
	VAR_INPUT
		nThickness	:	DINT;	(* Line thickness (if negative, the rectangle is filled) *)
		hrPrev	:	HRESULT;	(* HRESULT indicating the result of previous operations (If SUCCEEDED(hrPrev) equals false, no operation is executed.) *)
	END_VAR

END_FUNCTION

// Functions/Drawing/F_VN_DrawRectangle_TcVnRectangle_UDINT

	{attribute 'TcIecLibraryType'}
	{attribute 'external_name' := 'F_VN_DrawRectangle_TcVnRectangle_UDINT_GUID_537FBDE5_4020_27F8_65D4_084FE8AF7342'}
	(* Draw a rectangle. *)
	FUNCTION F_VN_DrawRectangle_TcVnRectangle_UDINT : HRESULT
	VAR_IN_OUT
		stRectangle	:	TcVnRectangle_UDINT;	(* Rectangle to be drawn *)
	END_VAR
	VAR_INPUT
		ipDestImage	:	ITcVnImage;	(* Destination image *)
	END_VAR
	VAR_IN_OUT
		aColor	:	TcVnVector4_LREAL;	(* Color *)
	END_VAR
	VAR_INPUT
		nThickness	:	DINT;	(* Line thickness (if negative, the rectangle is filled) *)
		hrPrev	:	HRESULT;	(* HRESULT indicating the result of previous operations (If SUCCEEDED(hrPrev) equals false, no operation is executed.) *)
	END_VAR

END_FUNCTION

// Functions/Drawing/F_VN_DrawRotatedRectangle

	{attribute 'TcIecLibraryType'}
	{attribute 'external_name' := 'F_VN_DrawRotatedRectangle_GUID_F1125FE7_F11E_21EE_550F_6DF6FDF001CD'}
	(* Draw a rectangle. *)
	FUNCTION F_VN_DrawRotatedRectangle : HRESULT
	VAR_IN_OUT
		stRectangle	:	TcVnRotatedRectangle;	(* Rectangle to be drawn (rotation angle in degrees) *)
	END_VAR
	VAR_INPUT
		ipDestImage	:	ITcVnImage;	(* Destination image *)
	END_VAR
	VAR_IN_OUT
		aColor	:	TcVnVector4_LREAL;	(* Color *)
	END_VAR
	VAR_INPUT
		nThickness	:	DINT;	(* Line thickness (if negative, the rectangle is filled) *)
		hrPrev	:	HRESULT;	(* HRESULT indicating the result of previous operations (If SUCCEEDED(hrPrev) equals false, no operation is executed.) *)
	END_VAR

END_FUNCTION

// Functions/Drawing/F_VN_DrawRotatedRectangleExp

	{attribute 'TcIecLibraryType'}
	{attribute 'external_name' := 'F_VN_DrawRotatedRectangleExp_GUID_E60B7262_090F_2C13_5EB0_4E7F85236119'}
	(* Draw a rectangle. (expert function) *)
	FUNCTION F_VN_DrawRotatedRectangleExp : HRESULT
	VAR_IN_OUT
		stRectangle	:	TcVnRotatedRectangle;	(* Rectangle to be drawn (rotation angle in degrees) *)
	END_VAR
	VAR_INPUT
		ipDestImage	:	ITcVnImage;	(* Destination image *)
	END_VAR
	VAR_IN_OUT
		aColor	:	TcVnVector4_LREAL;	(* Color *)
	END_VAR
	VAR_INPUT
		nThickness	:	DINT;	(* Line thickness (if negative, the rectangle is filled) *)
		eLineType	:	ETcVnLineType;	(* Line type *)
		hrPrev	:	HRESULT;	(* HRESULT indicating the result of previous operations (If SUCCEEDED(hrPrev) equals false, no operation is executed.) *)
	END_VAR

END_FUNCTION

// Functions/Drawing/F_VN_FillCircle

	{attribute 'TcIecLibraryType'}
	{attribute 'external_name' := 'F_VN_FillCircle_GUID_4FFA9EBC_743A_257E_6676_B381955FCAAB'}
	(* Paint a filled circle. *)
	FUNCTION F_VN_FillCircle : HRESULT
	VAR_INPUT
		nCenterX	:	UDINT;	(* x coordinate of the center *)
		nCenterY	:	UDINT;	(* y coordinate of the center *)
		nRadius	:	UDINT;	(* Radius *)
		ipDestImage	:	ITcVnImage;	(* Destination image *)
	END_VAR
	VAR_IN_OUT
		aColor	:	TcVnVector4_LREAL;	(* Color *)
	END_VAR
	VAR_INPUT
		hrPrev	:	HRESULT;	(* HRESULT indicating the result of previous operations (If SUCCEEDED(hrPrev) equals false, no operation is executed.) *)
	END_VAR

END_FUNCTION

// Functions/Drawing/F_VN_FillContours

	{attribute 'TcIecLibraryType'}
	{attribute 'external_name' := 'F_VN_FillContours_GUID_821A6D94_9653_2B5B_54A0_18C96BA3C198'}
	(* Paint a single point set or multiple point sets that are interpreted as contours. *)
	FUNCTION F_VN_FillContours : HRESULT
	VAR_INPUT
		ipContours	:	ITcVnContainer;	(* Single contour (ContainerType_Vector_TcVnPoint2_DINT) or multiple contours (ContainerType_Vector_Vector_TcVnPoint2_DINT) *)
		nContourIndex	:	DINT;	(* Index of a specific contour to be drawn (if negative, all contours within the container are drawn) *)
		ipDestImage	:	ITcVnImage;	(* Destination image *)
	END_VAR
	VAR_IN_OUT
		aColor	:	TcVnVector4_LREAL;	(* Color *)
	END_VAR
	VAR_INPUT
		hrPrev	:	HRESULT;	(* HRESULT indicating the result of previous operations (If SUCCEEDED(hrPrev) equals false, no operation is executed.) *)
	END_VAR

END_FUNCTION

// Functions/Drawing/F_VN_FillEllipse

	{attribute 'TcIecLibraryType'}
	{attribute 'external_name' := 'F_VN_FillEllipse_GUID_44D42548_1B41_20F1_5FD9_1318322D9492'}
	(* Paint a filled ellipse. *)
	FUNCTION F_VN_FillEllipse : HRESULT
	VAR_IN_OUT
		stEllipse	:	TcVnRotatedRectangle;	(* Ellipse to be painted (rotation angle in degrees) *)
	END_VAR
	VAR_INPUT
		ipDestImage	:	ITcVnImage;	(* Destination image *)
	END_VAR
	VAR_IN_OUT
		aColor	:	TcVnVector4_LREAL;	(* Color *)
	END_VAR
	VAR_INPUT
		hrPrev	:	HRESULT;	(* HRESULT indicating the result of previous operations (If SUCCEEDED(hrPrev) equals false, no operation is executed.) *)
	END_VAR

END_FUNCTION

// Functions/Drawing/F_VN_FillPolygon

	{attribute 'TcIecLibraryType'}
	{attribute 'external_name' := 'F_VN_FillPolygon_GUID_3DC658DB_99FA_201B_452C_8EB1D3BEFC8B'}
	(* Paint a filled pologon using a set of points. *)
	FUNCTION F_VN_FillPolygon : HRESULT
	VAR_INPUT
		ipPoints	:	ITcVnContainer;	(* Container with TcVnPoint2_DINT, TcVnPoint2_REAL, or TcVnPoint2_LREAL elements *)
		ipDestImage	:	ITcVnImage;	(* Destination image *)
	END_VAR
	VAR_IN_OUT
		aColor	:	TcVnVector4_LREAL;	(* Color *)
	END_VAR
	VAR_INPUT
		hrPrev	:	HRESULT;	(* HRESULT indicating the result of previous operations (If SUCCEEDED(hrPrev) equals false, no operation is executed.) *)
	END_VAR

END_FUNCTION

// Functions/Drawing/F_VN_FillRectangle

	{attribute 'TcIecLibraryType'}
	{attribute 'external_name' := 'F_VN_FillRectangle_GUID_AEFBF966_CDFD_251C_636A_00BA24CFACAB'}
	(* Paint a filled rectangle. *)
	FUNCTION F_VN_FillRectangle : HRESULT
	VAR_INPUT
		nTopLeftX	:	UDINT;	(* x coordinate of the top left corner *)
		nTopLeftY	:	UDINT;	(* y coordinate of the top left corner *)
		nBottomRightX	:	UDINT;	(* x coordinate of the bottom right corner *)
		nBottomRightY	:	UDINT;	(* y coordinate of the bottom right corner *)
		ipDestImage	:	ITcVnImage;	(* Destination image *)
	END_VAR
	VAR_IN_OUT
		aColor	:	TcVnVector4_LREAL;	(* Color *)
	END_VAR
	VAR_INPUT
		hrPrev	:	HRESULT;	(* HRESULT indicating the result of previous operations (If SUCCEEDED(hrPrev) equals false, no operation is executed.) *)
	END_VAR

END_FUNCTION

// Functions/Drawing/F_VN_FillRotatedRectangle

	{attribute 'TcIecLibraryType'}
	{attribute 'external_name' := 'F_VN_FillRotatedRectangle_GUID_1D162686_C5B0_27FF_5F59_A7E821AE31BC'}
	(* Paint a filled rectangle. *)
	FUNCTION F_VN_FillRotatedRectangle : HRESULT
	VAR_IN_OUT
		stRectangle	:	TcVnRotatedRectangle;	(* Rectangle to be painted (rotation angle in degrees) *)
	END_VAR
	VAR_INPUT
		ipDestImage	:	ITcVnImage;	(* Destination image *)
	END_VAR
	VAR_IN_OUT
		aColor	:	TcVnVector4_LREAL;	(* Color *)
	END_VAR
	VAR_INPUT
		hrPrev	:	HRESULT;	(* HRESULT indicating the result of previous operations (If SUCCEEDED(hrPrev) equals false, no operation is executed.) *)
	END_VAR

END_FUNCTION

// Functions/Drawing/F_VN_PlotIntensityProfile

	{attribute 'TcIecLibraryType'}
	{attribute 'external_name' := 'F_VN_PlotIntensityProfile_GUID_AAADF02B_4346_2BBF_472A_43CDCB738D01'}
	(* Plots the pixel intensity profile along a line segment in an image. *)
	FUNCTION F_VN_PlotIntensityProfile : HRESULT
	VAR_INPUT
		ipSrcImage	:	ITcVnImage;	(* Source image (USINT, 1 channel) *)
		ipDestImage	:	REFERENCE TO ITcVnImage;	(* Destination image (USINT, 1 channel. x: position, y: intensity, origin: bottom left. An appropriate destination image will be created if required.) *)
	END_VAR
	VAR_IN_OUT
		aStartPoint	:	TcVnPoint2_REAL;	(* Start point of the line segment *)
		aEndPoint	:	TcVnPoint2_REAL;	(* End point of the line segment *)
	END_VAR
	VAR_INPUT
		hrPrev	:	HRESULT;	(* HRESULT indicating the result of previous operations (If SUCCEEDED(hrPrev) equals false, no operation is executed.) *)
	END_VAR

END_FUNCTION

// Functions/Drawing/F_VN_PlotIntensityProfileExp

	{attribute 'TcIecLibraryType'}
	{attribute 'external_name' := 'F_VN_PlotIntensityProfileExp_GUID_00D19E72_3BC8_2C13_54A8_8D4B18C13213'}
	(* Plots the pixel intensity profile along a line segment in an image. (expert function) *)
	FUNCTION F_VN_PlotIntensityProfileExp : HRESULT
	VAR_INPUT
		ipSrcImage	:	ITcVnImage;	(* Source image (USINT, 1 channel) *)
		ipDestImage	:	REFERENCE TO ITcVnImage;	(* Destination image (USINT, 1 channel. x: position, y: intensity, origin: bottom left. An appropriate destination image will be created if required.) *)
	END_VAR
	VAR_IN_OUT
		aStartPoint	:	TcVnPoint2_REAL;	(* Start point of the line segment *)
		aEndPoint	:	TcVnPoint2_REAL;	(* End point of the line segment *)
		aBackgroundColor	:	TcVnVector4_LREAL;	(* Background color *)
		aLineColor	:	TcVnVector4_LREAL;	(* Line color *)
		aGridColor	:	TcVnVector4_LREAL;	(* Grid color *)
	END_VAR
	VAR_INPUT
		nScaleX	:	DINT;	(* Scale in x direction (ipDestImage will have a width of nScaleX * (ipSrcImage width - 1) + 1) *)
		nScaleY	:	DINT;	(* Scale in y direction (ipDestImage will have a height of nScaleY * 255 + 1) *)
		nThickness	:	DINT;	(* Line thickness *)
		nDestChannels	:	DINT;	(* ipDestImage channels (1 or 3) *)
		hrPrev	:	HRESULT;	(* HRESULT indicating the result of previous operations (If SUCCEEDED(hrPrev) equals false, no operation is executed.) *)
	END_VAR

END_FUNCTION

// Functions/Drawing/F_VN_PutLabel

	{attribute 'TcIecLibraryType'}
	{attribute 'external_name' := 'F_VN_PutLabel_GUID_B42C8837_CD3F_241B_5A2A_689EC24150BE'}
	(* Write a label (black text on white background) into an image. *)
	FUNCTION F_VN_PutLabel : HRESULT
	VAR_IN_OUT CONSTANT
		sText	:	STRING;	(* Text *)
	END_VAR
	VAR_INPUT
		ipDestImage	:	ITcVnImage;	(* Destination image *)
		nX	:	UDINT;	(* x coordinate (bottom left) *)
		nY	:	UDINT;	(* y coordinate (bottom left) *)
		fFontScale	:	LREAL;	(* Scaling factor *)
		hrPrev	:	HRESULT;	(* HRESULT indicating the result of previous operations (If SUCCEEDED(hrPrev) equals false, no operation is executed.) *)
	END_VAR

END_FUNCTION

// Functions/Drawing/F_VN_PutLabelExp

	{attribute 'TcIecLibraryType'}
	{attribute 'external_name' := 'F_VN_PutLabelExp_GUID_3AD8E894_0BC4_259B_7CA7_3DE9674556FD'}
	(* Write a label (text on unified background) into an image. (expert function) *)
	FUNCTION F_VN_PutLabelExp : HRESULT
	VAR_IN_OUT CONSTANT
		sText	:	STRING;	(* Text *)
	END_VAR
	VAR_INPUT
		ipDestImage	:	ITcVnImage;	(* Destination image *)
		nX	:	UDINT;	(* x coordinate (bottom left) *)
		nY	:	UDINT;	(* y coordinate (bottom left) *)
		fFontScale	:	LREAL;	(* Scaling factor *)
		nThickness	:	UDINT;	(* Line thickness *)
		eFontType	:	ETcVnFontType;	(* Font type *)
	END_VAR
	VAR_IN_OUT
		aFontColor	:	TcVnVector4_LREAL;	(* Font color *)
		aBackgroundColor	:	TcVnVector4_LREAL;	(* Background color *)
	END_VAR
	VAR_INPUT
		eLineType	:	ETcVnLineType;	(* Line type *)
		hrPrev	:	HRESULT;	(* HRESULT indicating the result of previous operations (If SUCCEEDED(hrPrev) equals false, no operation is executed.) *)
	END_VAR

END_FUNCTION

// Functions/Drawing/F_VN_PutText

	{attribute 'TcIecLibraryType'}
	{attribute 'external_name' := 'F_VN_PutText_GUID_9289C3DD_0299_2B45_5BF4_875BAA264BBE'}
	(* Write text into an image. *)
	FUNCTION F_VN_PutText : HRESULT
	VAR_IN_OUT CONSTANT
		sText	:	STRING;	(* Text *)
	END_VAR
	VAR_INPUT
		ipDestImage	:	ITcVnImage;	(* Destination image *)
		nX	:	UDINT;	(* x coordinate (bottom left) *)
		nY	:	UDINT;	(* y coordinate (bottom left) *)
		eFontType	:	ETcVnFontType;	(* Font type *)
		fFontScale	:	LREAL;	(* Scaling factor *)
	END_VAR
	VAR_IN_OUT
		aColor	:	TcVnVector4_LREAL;	(* Text color *)
	END_VAR
	VAR_INPUT
		hrPrev	:	HRESULT;	(* HRESULT indicating the result of previous operations (If SUCCEEDED(hrPrev) equals false, no operation is executed.) *)
	END_VAR

END_FUNCTION

// Functions/Drawing/F_VN_PutTextExp

	{attribute 'TcIecLibraryType'}
	{attribute 'external_name' := 'F_VN_PutTextExp_GUID_C080A95A_603B_2592_679E_8B8B8D0BED94'}
	(* Write text into an image. (expert function) *)
	FUNCTION F_VN_PutTextExp : HRESULT
	VAR_IN_OUT CONSTANT
		sText	:	STRING;	(* Text *)
	END_VAR
	VAR_INPUT
		ipDestImage	:	ITcVnImage;	(* Destination image *)
		nX	:	UDINT;	(* x coordinate (bottom left) *)
		nY	:	UDINT;	(* y coordinate (bottom left) *)
		eFontType	:	ETcVnFontType;	(* Font type *)
		fFontScale	:	LREAL;	(* Scaling factor *)
	END_VAR
	VAR_IN_OUT
		aColor	:	TcVnVector4_LREAL;	(* Text color *)
	END_VAR
	VAR_INPUT
		nThickness	:	DINT;	(* Line thickness *)
		eLineType	:	ETcVnLineType;	(* Line type *)
		bBottomLeftOrigin	:	BOOL;	(* Sets the image origin to the bottom left corner, if true *)
		hrPrev	:	HRESULT;	(* HRESULT indicating the result of previous operations (If SUCCEEDED(hrPrev) equals false, no operation is executed.) *)
	END_VAR

END_FUNCTION

// Functions/Neural Network/F_VN_ConvertDataLayout

	{attribute 'TcIecLibraryType'}
	{attribute 'external_name' := 'F_VN_ConvertDataLayout_GUID_21981C8F_19DA_2DDF_62A9_1D4DBD7E13CC'}
	(* Convert a data layout (the arrangement of dimensions in the input data) to another data layout. *)
	FUNCTION F_VN_ConvertDataLayout : HRESULT
	VAR_INPUT
		ipSrcImage	:	ITcVnImage;	(* Source image *)
		ipDestImage	:	REFERENCE TO ITcVnImage;	(* Destination image (An appropriate destination image will be created if required.) *)
		nSrcDataLayout	:	ULINT;	(* Data layout of the source image (Commonly used data layouts are available in the enumeration ETcVnDataLayout. If nSrcDataLayout is set to 0 or TCVN_DL_DEFAULT, the DataLayout will be automatically determined based on the dimension of the ipSrcImage: 0x12 for 2D, 0x123 for 3D, 0x1234 for 4D, and so forth.) *)
		nDestDataLayout	:	ULINT;	(* Required output data layout (Commonly used data layouts are available in the enumeration ETcVnDataLayout. nDestDataLayout must not equal 0 or TCVN_DL_DEFAULT.) *)
		hrPrev	:	HRESULT;	(* HRESULT indicating the result of previous operations (If SUCCEEDED(hrPrev) equals false, no operation is executed.) *)
	END_VAR

END_FUNCTION

// Functions/Neural Network/F_VN_ReshapeImage

	{attribute 'TcIecLibraryType'}
	{attribute 'external_name' := 'F_VN_ReshapeImage_GUID_33B79AA7_4730_275F_45C8_977CCA382433'}
	(* Changes the shape of an ITcVnImage. The total number of elements in the new shape must be equal to the total number of elements in ipSrcImage. *)
	FUNCTION F_VN_ReshapeImage : HRESULT
	VAR_INPUT
		ipSrcImage	:	ITcVnImage;	(* Source image (1 channel) *)
		ipDestImage	:	REFERENCE TO ITcVnImage;	(* Destination image (An appropriate single channel destination image will be created if required.) *)
	END_VAR
	VAR_IN_OUT
		aNewShape	:	TcVnArray33_UDINT;	(* Specifies the shape of ipDestImage. First entry is the number of dimensions (max. 32), followed by the sizes of each dimension. If one dimension is set to zero, its value will be automatically calculated based on the total elements of ipSrcImage (Only one dimension can be set to zero.) *)
	END_VAR
	VAR_INPUT
		hrPrev	:	HRESULT;	(* HRESULT indicating the result of previous operations (If SUCCEEDED(hrPrev) equals false, no operation is executed.) *)
	END_VAR

END_FUNCTION

// Functions/Neural Network/F_VN_Sigmoid

	{attribute 'TcIecLibraryType'}
	{attribute 'external_name' := 'F_VN_Sigmoid_GUID_5C335F46_61F7_2834_4D32_F097D4F6D65F'}
	(* Apply the standard logistic function 1 / (1 + exp(-x)) element-wise to a single- or multi-channel REAL image. *)
	FUNCTION F_VN_Sigmoid : HRESULT
	VAR_INPUT
		ipSrcImage	:	ITcVnImage;	(* Source image (REAL) *)
		ipDestImage	:	REFERENCE TO ITcVnImage;	(* Destination image (An appropriate destination image will be created if required.) *)
		hrPrev	:	HRESULT;	(* HRESULT indicating the result of previous operations (If SUCCEEDED(hrPrev) equals false, no operation is executed.) *)
	END_VAR

END_FUNCTION

// Functions/Neural Network/F_VN_SigmoidExp

	{attribute 'TcIecLibraryType'}
	{attribute 'external_name' := 'F_VN_SigmoidExp_GUID_AE577732_3D07_272A_7D23_DC3E2A2104C4'}
	(* Apply the logistic function 1 / (1 + exp(-fSteepness * (x - fShift))) element-wise to a single- or multi-channel REAL image. (expert function) *)
	FUNCTION F_VN_SigmoidExp : HRESULT
	VAR_INPUT
		ipSrcImage	:	ITcVnImage;	(* Source image (REAL) *)
		ipDestImage	:	REFERENCE TO ITcVnImage;	(* Destination image (An appropriate destination image will be created if required.) *)
		fShift	:	REAL;	(* Determines the intensity level around which the logistic function transitions. *)
		fSteepness	:	REAL;	(* Controls the sharpness of the transition. *)
		hrPrev	:	HRESULT;	(* HRESULT indicating the result of previous operations (If SUCCEEDED(hrPrev) equals false, no operation is executed.) *)
	END_VAR

END_FUNCTION

// Functions/Neural Network/F_VN_SoftMax

	{attribute 'TcIecLibraryType'}
	{attribute 'external_name' := 'F_VN_SoftMax_GUID_7AACE923_07E1_29BA_6A0B_5E0012C2EF14'}
	(* Apply softmax function pixel-wise to a single channel REAL image. *)
	FUNCTION F_VN_SoftMax : HRESULT
	VAR_INPUT
		ipSrcImage	:	ITcVnImage;	(* Source image (REAL, 1 channel) *)
		ipDestImage	:	REFERENCE TO ITcVnImage;	(* Destination image (An appropriate single channel destination image will be created if required.) *)
		bFlatten	:	BOOL;	(* If true, the resulting image will be reshaped into a single row. *)
		hrPrev	:	HRESULT;	(* HRESULT indicating the result of previous operations (If SUCCEEDED(hrPrev) equals false, no operation is executed.) *)
	END_VAR

END_FUNCTION

// Functions/Neural Network/F_VN_NonMaxSuppression

	{attribute 'TcIecLibraryType'}
	{attribute 'external_name' := 'F_VN_NonMaxSuppression_GUID_C5DBABC7_B34E_2892_4BC4_87DC2E004E6A'}
	(* Perform non-maximum suppression on given bounding boxes and corresponding scores. *)
	FUNCTION F_VN_NonMaxSuppression : HRESULT
	VAR_INPUT
		ipBoundingBoxes	:	ITcVnContainer;	(* Container of bounding boxes to apply the non maximum supresion (ContainerType_Vector_TcVnRectangle_DINT) *)
		ipScores	:	ITcVnContainer;	(* Container of coreeponding score for each bounding box (ContainerType_Vector_REAL) *)
		ipDestIndcies	:	REFERENCE TO ITcVnContainer;	(* Container of the kept indcies after apply the non maximum suppression (ContainerType_Vector_DINT) *)
		fScoreThreshold	:	REAL;	(* A threshold [0.0 to 1.0] used to filter the bounding boxes by score *)
		fOverlapThreshold	:	REAL;	(* A threshold [0.0 to 1.0] that determines the minimum degree of intersection over union (IoU) required for bounding boxes to be considered overlapping *)
		hrPrev	:	HRESULT;	(* HRESULT indicating the result of previous operations (If SUCCEEDED(hrPrev) equals false, no operation is executed.) *)
	END_VAR

END_FUNCTION

// Functions/Neural Network/F_VN_NonMaxSuppressionExp

	{attribute 'TcIecLibraryType'}
	{attribute 'external_name' := 'F_VN_NonMaxSuppressionExp_GUID_3D4EB8C2_75AD_21C3_67DE_761E06C1B05E'}
	(* Perform non-maximum suppression on given bounding boxes and corresponding scores. (expert function) *)
	FUNCTION F_VN_NonMaxSuppressionExp : HRESULT
	VAR_INPUT
		ipBoundingBoxes	:	ITcVnContainer;	(* Container of bounding boxes to apply the non maximum supresion (ContainerType_Vector_TcVnRectangle_DINT) *)
		ipScores	:	ITcVnContainer;	(* Container of coreeponding score for each bounding box (ContainerType_Vector_REAL) *)
		ipDestIndcies	:	REFERENCE TO ITcVnContainer;	(* Container of the kept indcies after apply the non maximum suppression (ContainerType_Vector_DINT) *)
		fScoreThreshold	:	REAL;	(* A threshold [0.0 to 1.0] used to filter the bounding boxes by score *)
		fOverlapThreshold	:	REAL;	(* A threshold [0.0 to 1.0] that determines the minimum degree of intersection over union (IoU) required for bounding boxes to be considered overlapping *)
		ipClassIndcies	:	ITcVnContainer;	(* Container of corresponding set of class indcies (ContainerType_Vector_DINT) *)
		fEta	:	REAL;	(* An adjustable threshold [0.0 to 1.0] used to dynamically reduce the overlap threshold during processing. Setting it to 1 maintains a constant value for the overlap threshold *)
		nTopK	:	DINT;	(* The maximum number of bounding boxes with the highest scores to undergo the suppression algorithm (must be >= 0). Setting it to zero applies the algorithm to all bounding boxes *)
		hrPrev	:	HRESULT;	(* HRESULT indicating the result of previous operations (If SUCCEEDED(hrPrev) equals false, no operation is executed.) *)
	END_VAR

END_FUNCTION

// Functions/Neural Network/F_VN_ExecuteNeuralNetwork

	{attribute 'TcIecLibraryType'}
	{attribute 'external_name' := 'F_VN_ExecuteNeuralNetwork_GUID_797DBC99_F393_2420_4950_B14ED43E9BED'}
	(* Execute a neural network using the provided image as input and provide the output of one output layer. The function doesn't perform any pre-processing or transformation. *)
	FUNCTION F_VN_ExecuteNeuralNetwork : HRESULT
	VAR_INPUT
		ipNeuralNetwork	:	ITcVnNeuralNetwork;	(* Neural network model *)
		ipSrcImage	:	ITcVnImage;	(* Source image (The image layout must be adapted to match the model's expected input format using e.g. F_VN_ConvertDataLayout or F_VN_ReshapeImage functions if necessary.) *)
		ipDestImage	:	REFERENCE TO ITcVnImage;	(* Destination image (An appropriate destination image based on the output layer is created. To process the destination image, use e.g. F_VN_ConvertDataLayout or F_VN_ReshapeImage if necessary. *)
		hrPrev	:	HRESULT;	(* HRESULT indicating the result of previous operations (If SUCCEEDED(hrPrev) equals false, no operation is executed.) *)
	END_VAR

END_FUNCTION

// Functions/Neural Network/F_VN_ExecuteNeuralNetwork_MI

	{attribute 'TcIecLibraryType'}
	{attribute 'external_name' := 'F_VN_ExecuteNeuralNetwork_MI_GUID_A1EF92AA_206B_2C21_67C3_E72D98047F52'}
	(* Execute a neural network with multiple inputs (MI) using the provided images. Ensure all model input names are listed in sInputNames and that the images and names are in the same order. The result of one output layer is returned. The function doesn't perform any pre-processing or transformation. *)
	FUNCTION F_VN_ExecuteNeuralNetwork_MI : HRESULT
	VAR_INPUT
		ipNeuralNetwork	:	ITcVnNeuralNetwork;	(* Neural network model *)
		pSrcImages	:	PVOID;	(* Pointer to an array of source input images *)
		nSrcArraySize	:	UINT;	(* The size of the array referenced by pSrcImages. pSrcImages must reference an array with a size equal to the number of model inputs. *)
	END_VAR
	VAR_IN_OUT CONSTANT
		sInputNames	:	STRING;	(* Input names separated by ";" *)
	END_VAR
	VAR_INPUT
		ipDestImage	:	REFERENCE TO ITcVnImage;	(* Destination image (An appropriate destination image based on the output layer is created. To process the destination image, use e.g. F_VN_ConvertDataLayout or F_VN_ReshapeImage if necessary. *)
		hrPrev	:	HRESULT;	(* HRESULT indicating the result of previous operations (If SUCCEEDED(hrPrev) equals false, no operation is executed.) *)
	END_VAR

END_FUNCTION

// Functions/Neural Network/F_VN_ExecuteNeuralNetwork_MultiLayerOutput

	{attribute 'TcIecLibraryType'}
	{attribute 'external_name' := 'F_VN_ExecuteNeuralNetwork_MultiLayerOutput_GUID_DDC222CE_1B06_2011_6D73_D1126BEC91D4'}
	(* This function is deprecated, please use F_VN_ExecuteNeuralNetwork_MO. Execute a neural network using the provided image as input and provide the output of the specified output layers. The function doesn't perform any pre-processing or transformation. *)
	FUNCTION F_VN_ExecuteNeuralNetwork_MultiLayerOutput : HRESULT
	VAR_INPUT
		ipNeuralNetwork	:	ITcVnNeuralNetwork;	(* Neural network model *)
		ipSrcImage	:	ITcVnImage;	(* Source image (The image layout must be adapted to match the model's expected input format using e.g. F_VN_ConvertDataLayout or F_VN_ReshapeImage functions if necessary.) *)
		ipDestImages	:	REFERENCE TO ITcVnContainer;	(* Container of images containing the output from the specified layers. *)
		ipLayerNames	:	ITcVnContainer;	(* Container of layer names whose outputs to be returned (ContainerType_Vector_String_SINT). If set to zero, the outputs of all unconnected output layers will be returned.. *)
		hrPrev	:	HRESULT;	(* HRESULT indicating the result of previous operations (If SUCCEEDED(hrPrev) equals false, no operation is executed.) *)
	END_VAR

END_FUNCTION

// Functions/Neural Network/F_VN_ExecuteNeuralNetwork_MO

	{attribute 'TcIecLibraryType'}
	{attribute 'external_name' := 'F_VN_ExecuteNeuralNetwork_MO_GUID_72FEEABA_2B32_2A3D_5342_75F9CA3FE8B7'}
	(* Execute a neural network using the provided image as input and provide the output of the specified output layers. The function doesn't perform any pre-processing or transformation. *)
	FUNCTION F_VN_ExecuteNeuralNetwork_MO : HRESULT
	VAR_INPUT
		ipNeuralNetwork	:	ITcVnNeuralNetwork;	(* Neural network model *)
		ipSrcImage	:	ITcVnImage;	(* Source image (The image layout must be adapted to match the model's expected input format using e.g. F_VN_ConvertDataLayout or F_VN_ReshapeImage functions if necessary.) *)
		ipDestImages	:	REFERENCE TO ITcVnContainer;	(* Container of images containing the output from the specified layers. *)
		ipOutputNames	:	ITcVnContainer;	(* Container of layer names whose outputs to be returned (ContainerType_Vector_String_SINT). If set to zero, the outputs of all unconnected output layers will be returned.. *)
		hrPrev	:	HRESULT;	(* HRESULT indicating the result of previous operations (If SUCCEEDED(hrPrev) equals false, no operation is executed.) *)
	END_VAR

END_FUNCTION

// Functions/Neural Network/F_VN_ExecuteNeuralNetwork_MIMO_String

	{attribute 'TcIecLibraryType'}
	{attribute 'external_name' := 'F_VN_ExecuteNeuralNetwork_MIMO_String_GUID_612B98B8_D67D_2BBC_5E09_3393A5DDACD3'}
	(* Execute a neural network with multiple inputs and multiple outputs (MIMO) using the provided images. Ensure all model input names are listed in sInputNames and that the images and names are in the same order. The result of the specified output layers are returned. The function doesn't perform any pre-processing or transformation. *)
	FUNCTION F_VN_ExecuteNeuralNetwork_MIMO_String : HRESULT
	VAR_INPUT
		ipNeuralNetwork	:	ITcVnNeuralNetwork;	(* Neural network model *)
		pSrcImages	:	PVOID;	(* Pointer to an array of source input images *)
		nSrcArraySize	:	UINT;	(* The size of the array referenced by pSrcImages. pSrcImages must reference an array with a size equal to the number of model inputs. *)
	END_VAR
	VAR_IN_OUT CONSTANT
		sInputNames	:	STRING;	(* Input names separated by ";" *)
	END_VAR
	VAR_INPUT
		ipDestImages	:	REFERENCE TO ITcVnContainer;	(* Container of images containing the output from the specified layers. *)
	END_VAR
	VAR_IN_OUT CONSTANT
		sOutputNames	:	STRING;	(* Names of output layers whose outputs are required separated by ";". If empty, the outputs of all unconnected output layers are provided. *)
	END_VAR
	VAR_INPUT
		hrPrev	:	HRESULT;	(* HRESULT indicating the result of previous operations (If SUCCEEDED(hrPrev) equals false, no operation is executed.) *)
	END_VAR

END_FUNCTION

// Functions/Neural Network/F_VN_ExecuteNeuralNetwork_SingleLayerOutput

	{attribute 'TcIecLibraryType'}
	{attribute 'external_name' := 'F_VN_ExecuteNeuralNetwork_SingleLayerOutput_GUID_02844FE1_02C4_2B0F_6835_E22CD31F08A5'}
	(* This function is deprecated, please use F_VN_ExecuteNeuralNetwork_SO. Execute a neural network using the provided image as input and provide the output of the specified output layer. The function doesn't perform any pre-processing or transformation. *)
	FUNCTION F_VN_ExecuteNeuralNetwork_SingleLayerOutput : HRESULT
	VAR_INPUT
		ipNeuralNetwork	:	ITcVnNeuralNetwork;	(* Neural network model *)
		ipSrcImage	:	ITcVnImage;	(* Source image (The image layout must be adapted to match the model's expected input format using e.g. F_VN_ConvertDataLayout or F_VN_ReshapeImage functions if necessary.) *)
		ipDestImage	:	REFERENCE TO ITcVnImage;	(* Destination image (An appropriate destination image based on the output layer is created. To process the destination image, use e.g. F_VN_ConvertDataLayout or F_VN_ReshapeImage if necessary. *)
	END_VAR
	VAR_IN_OUT CONSTANT
		sLayerName	:	STRING;	(* Specify the name of the layer for which the output is required. If empty, the output of one output layer is provided. *)
	END_VAR
	VAR_INPUT
		hrPrev	:	HRESULT;	(* HRESULT indicating the result of previous operations (If SUCCEEDED(hrPrev) equals false, no operation is executed.) *)
	END_VAR

END_FUNCTION

// Functions/Neural Network/F_VN_ExecuteNeuralNetwork_SO

	{attribute 'TcIecLibraryType'}
	{attribute 'external_name' := 'F_VN_ExecuteNeuralNetwork_SO_GUID_B012F955_2AD7_2180_4719_71F04482E824'}
	(* Execute a neural network using the provided image as input and provide the output of the specified output layer. The function doesn't perform any pre-processing or transformation. *)
	FUNCTION F_VN_ExecuteNeuralNetwork_SO : HRESULT
	VAR_INPUT
		ipNeuralNetwork	:	ITcVnNeuralNetwork;	(* Neural network model *)
		ipSrcImage	:	ITcVnImage;	(* Source image (The image layout must be adapted to match the model's expected input format using e.g. F_VN_ConvertDataLayout or F_VN_ReshapeImage functions if necessary.) *)
		ipDestImage	:	REFERENCE TO ITcVnImage;	(* Destination image (An appropriate destination image based on the output layer is created. To process the destination image, use e.g. F_VN_ConvertDataLayout or F_VN_ReshapeImage if necessary. *)
	END_VAR
	VAR_IN_OUT CONSTANT
		sOutputName	:	STRING;	(* Specify the name of the layer for which the output is required. If empty, the output of one output layer is provided. *)
	END_VAR
	VAR_INPUT
		hrPrev	:	HRESULT;	(* HRESULT indicating the result of previous operations (If SUCCEEDED(hrPrev) equals false, no operation is executed.) *)
	END_VAR

END_FUNCTION

// Functions/Neural Network/F_VN_ExecuteNeuralNetwork_MISO

	{attribute 'TcIecLibraryType'}
	{attribute 'external_name' := 'F_VN_ExecuteNeuralNetwork_MISO_GUID_D763B0C7_8D60_2F73_4E94_3844642997A9'}
	(* Execute a neural network with multiple inputs and single output (MISO) using the provided images. Ensure all model input names are listed in sInputNames and that the images and names are in the same order. The result of the specified output layer is returned. The function doesn't perform any pre-processing or transformation. *)
	FUNCTION F_VN_ExecuteNeuralNetwork_MISO : HRESULT
	VAR_INPUT
		ipNeuralNetwork	:	ITcVnNeuralNetwork;	(* Neural network model *)
		pSrcImages	:	PVOID;	(* Pointer to an array of source input images *)
		nSrcArraySize	:	UINT;	(* The size of the array referenced by pSrcImages. pSrcImages must reference an array with a size equal to the number of model inputs. *)
	END_VAR
	VAR_IN_OUT CONSTANT
		sInputNames	:	STRING;	(* Input names separated by ";" *)
	END_VAR
	VAR_INPUT
		ipDestImage	:	REFERENCE TO ITcVnImage;	(* Destination image (An appropriate destination image based on the output layer is created. To process the destination image, use e.g. F_VN_ConvertDataLayout or F_VN_ReshapeImage if necessary. *)
	END_VAR
	VAR_IN_OUT CONSTANT
		sOutputName	:	STRING;	(* Specify the name of the layer for which the output is required. If empty, the output of one output layer is provided. *)
	END_VAR
	VAR_INPUT
		hrPrev	:	HRESULT;	(* HRESULT indicating the result of previous operations (If SUCCEEDED(hrPrev) equals false, no operation is executed.) *)
	END_VAR

END_FUNCTION

// Functions/Neural Network/F_VN_GetNeuralNetworkLayerNames

	{attribute 'TcIecLibraryType'}
	{attribute 'external_name' := 'F_VN_GetNeuralNetworkLayerNames_GUID_3A36A3D5_29D6_2E41_66F1_5A0EA497B03E'}
	(* Get the name of all layers in the neural network model. If the bOnlyOuput flag is set to true, only the unconnected output layer names are returned. *)
	FUNCTION F_VN_GetNeuralNetworkLayerNames : HRESULT
	VAR_INPUT
		ipNeuralNetwork	:	ITcVnNeuralNetwork;	(* Neural network model *)
		ipLayerNames	:	REFERENCE TO ITcVnContainer;	(* Container with the layers names (ContainerType_Vector_String_SINT)  *)
		bOnlyOutputs	:	BOOL;	(* If true, only the unconnected output layer names are returned. *)
		hrPrev	:	HRESULT;	(* HRESULT indicating the result of previous operations (If SUCCEEDED(hrPrev) equals false, no operation is executed.) *)
	END_VAR

END_FUNCTION

// Functions/Neural Network/F_VN_GetNeuralNetworkLayerNamesExp

	{attribute 'TcIecLibraryType'}
	{attribute 'external_name' := 'F_VN_GetNeuralNetworkLayerNamesExp_GUID_7BC9DA6B_5AEA_2C28_45C2_6540C58DDAED'}
	(* Get the name of model layers in the neural network model. (expert function) *)
	FUNCTION F_VN_GetNeuralNetworkLayerNamesExp : HRESULT
	VAR_INPUT
		ipNeuralNetwork	:	ITcVnNeuralNetwork;	(* Neural network model *)
		ipLayerNames	:	REFERENCE TO ITcVnContainer;	(* Container with the layers names (ContainerType_Vector_String_SINT) *)
		eLayerNameType	:	ETcVnLayerNameType;	(* Layer name type *)
		hrPrev	:	HRESULT;	(* HRESULT indicating the result of previous operations (If SUCCEEDED(hrPrev) equals false, no operation is executed.) *)
	END_VAR

END_FUNCTION

// Functions/Neural Network/F_VN_GetNeuralNetworkLayerNamesExp_String

	{attribute 'TcIecLibraryType'}
	{attribute 'external_name' := 'F_VN_GetNeuralNetworkLayerNamesExp_String_GUID_95E73A2C_6035_2E1F_68C1_B56DEF857B8F'}
	(* Get the name of model layers in the neural network model. (expert function) *)
	FUNCTION F_VN_GetNeuralNetworkLayerNamesExp_String : HRESULT
	VAR_INPUT
		ipNeuralNetwork	:	ITcVnNeuralNetwork;	(* Neural network model *)
	END_VAR
	VAR_IN_OUT CONSTANT
		sLayerNames	:	STRING;	(* Layer names separated by ";". Make sure to choose a sufficient STRING size! *)
	END_VAR
	VAR_INPUT
		nMaxLength	:	ULINT;	(* Maximum string length to export (including 0 termination). If the container content is longer, the string is cut off at nMaxLength - 1 and 0 termination is appended. In this case, S_FALSE is returned. *)
		eLayerNameType	:	ETcVnLayerNameType;	(* Layer name type *)
		hrPrev	:	HRESULT;	(* HRESULT indicating the result of previous operations (If SUCCEEDED(hrPrev) equals false, no operation is executed.) *)
	END_VAR

END_FUNCTION

// Functions/Neural Network/F_VN_Reduce

	{attribute 'TcIecLibraryType'}
	{attribute 'external_name' := 'F_VN_Reduce_GUID_7BBAD4F1_D8C2_2BB5_6150_8C19FF4DDB1A'}
	(* Reduce ipSrcImage by applying the specified operation across rows/columns to obtain a single row/column/channel with the resulting values. *)
	FUNCTION F_VN_Reduce : HRESULT
	VAR_INPUT
		ipSrcImage	:	ITcVnImage;	(* Source image (USINT or REAL elements, 1 channel) *)
		ipDestImage	:	REFERENCE TO ITcVnImage;	(* Destination image. If ipSrcImage is of type USINT and the reduction type is SUM or AVG, ipDestImage will be of type REAL; otherwise, it retains the same type as ipSrcImage (An appropriate single channel destination image will be created if required.) *)
		nDim	:	DINT;	(* Index along which the ITcVnImage is reduced: 0 reduces the matrix to a single row, 1 reduces it to a single column, and 2 reduces to a single channel *)
		eReduceType	:	ETcVnReduceType;	(* Reduction operation *)
		hrPrev	:	HRESULT;	(* HRESULT indicating the result of previous operations (If SUCCEEDED(hrPrev) equals false, no operation is executed.) *)
	END_VAR

END_FUNCTION

// Functions/Neural Network/F_VN_ReduceArg

	{attribute 'TcIecLibraryType'}
	{attribute 'external_name' := 'F_VN_ReduceArg_GUID_9C3593E7_3AE1_26FE_7AF2_10CEE02A0D8B'}
	(* Finds indices of max/min elements along provided axis and reduce the ipSrcImage to a single row/column/channel. *)
	FUNCTION F_VN_ReduceArg : HRESULT
	VAR_INPUT
		ipSrcImage	:	ITcVnImage;	(* Source image *)
		ipDestImage	:	REFERENCE TO ITcVnImage;	(* Destination image of type DINT (An appropriate single channel destination image will be created if required.) *)
		nDim	:	DINT;	(* Index along which the ipSrcImage is reduced: 0 reduces the matrix to a single row, 1 reduces it to a single column, and 2 reduces to a single channel *)
		eReduceType	:	DINT;	(* Reduction operation REDUCE_MAX or REDUCE_MIN *)
		hrPrev	:	HRESULT;	(* HRESULT indicating the result of previous operations (If SUCCEEDED(hrPrev) equals false, no operation is executed.) *)
	END_VAR

END_FUNCTION

// Functions/Keypoint Features/F_VN_FilterGoodMatches

	{attribute 'TcIecLibraryType'}
	{attribute 'external_name' := 'F_VN_FilterGoodMatches_GUID_07AD8C34_B721_205D_74B5_D36ECCF07D96'}
	(* Filter the descriptor matches and return only good ones. *)
	FUNCTION F_VN_FilterGoodMatches : HRESULT
	VAR_INPUT
		ipMatches	:	ITcVnContainer;	(* Container with descriptor matches (ContainerType_Vector_TcVnDMatch or ContainerType_Vector_Vector_TcVnDMatch) *)
		ipGoodMatches	:	REFERENCE TO ITcVnContainer;	(* Returns a container with good matches (ContainerType_Vector_TcVnDMatch) *)
		fMaxDist	:	REAL;	(* Maximum allowed descriptor distance (-1 disables this filter criterion) *)
		fMaxKnnRatio	:	REAL;	(* Maximum allowed distance ratio between first and second best match ([0..1], used for knn match results only, -1 disables this filter criterion) *)
		hrPrev	:	HRESULT;	(* HRESULT indicating the result of previous operations (If SUCCEEDED(hrPrev) equals false, no operation is executed.) *)
	END_VAR

END_FUNCTION

// Functions/Keypoint Features/F_VN_FindReferenceKeyPointsInImage

	{attribute 'TcIecLibraryType'}
	{attribute 'external_name' := 'F_VN_FindReferenceKeyPointsInImage_GUID_06F4087C_9C8D_2632_6D2B_01DC94789DB8'}
	(* Searches a reference image, represented by its keypoints and corresponding descriptors, in a given source image. *)
	FUNCTION F_VN_FindReferenceKeyPointsInImage : HRESULT
	VAR_INPUT
		ipSrcKeyPoints	:	ITcVnContainer;	(* KeyPoints of the source image, e.g. (ContainerType_Vector_TcVnKeyPoint) *)
		ipSrcDescriptors	:	ITcVnImage;	(* Descriptors of the source image KeyPoints *)
		ipRefKeyPoints	:	ITcVnContainer;	(* KeyPoints of the reference image, e.g. (ContainerType_Vector_TcVnKeyPoint) *)
		ipRefDescriptors	:	ITcVnImage;	(* Descriptors of the reference image KeyPoints *)
		nRefImageWidth	:	UDINT;	(* Width of the reference image in pixels *)
		nRefImageHeight	:	UDINT;	(* Height of the reference image in pixels *)
		ipEdgePoints	:	REFERENCE TO ITcVnContainer;	(* Returns a container with the 4 edge points of the reference image transformed into the coordinates of the source image (ContainerType_Vector_TcVnPoint2_REAL) *)
		fMaxDist	:	REAL;	(* Maximum allowed descriptor distance (-1 disables this filter criterion) *)
		fMaxKnnRatio	:	REAL;	(* Maximum allowed distance ratio between first and second best match ([0..1], -1 disables this filter criterion) *)
		eNormType	:	ETcVnNormalizationType;	(* Normalization type used for descriptor matching (HAMMING recommended for AKAZE, ORB, and BRISK. HAMMING2 is recommended for ORB if the ORB nBriefPoints parameter is 3 or 4. ) *)
		hrPrev	:	HRESULT;	(* HRESULT indicating the result of previous operations (If SUCCEEDED(hrPrev) equals false, no operation is executed.) *)
	END_VAR
	VAR_OUTPUT
		aPerspectiveTransform	:	TcVnMatrix3x3_LREAL;	(* Returns the perspective transformation matrix, which transforms the reference points to the source points *)
		nNumberOfGoodMatches	:	UDINT;	(* Return the number of good matches *)
		nNumberOfInliers	:	UDINT;	(* Return the number of inlier matches *)
	END_VAR

END_FUNCTION

// Functions/Keypoint Features/F_VN_FindReferenceKeyPointsInImageExp

	{attribute 'TcIecLibraryType'}
	{attribute 'external_name' := 'F_VN_FindReferenceKeyPointsInImageExp_GUID_4297F7A3_B678_26F6_51BF_400E3F1145AA'}
	(* Searches a reference image, represented by its keypoints and corresponding descriptors, in a given source image. (expert function) *)
	FUNCTION F_VN_FindReferenceKeyPointsInImageExp : HRESULT
	VAR_INPUT
		ipSrcKeyPoints	:	ITcVnContainer;	(* KeyPoints of the source image, e.g. (ContainerType_Vector_TcVnKeyPoint) *)
		ipSrcDescriptors	:	ITcVnImage;	(* Descriptors of the source image KeyPoints *)
		ipRefKeyPoints	:	ITcVnContainer;	(* KeyPoints of the reference image (ContainerType_Vector_TcVnKeyPoint) *)
		ipRefDescriptors	:	ITcVnImage;	(* Descriptors of the reference image KeyPoints *)
		nRefImageWidth	:	UDINT;	(* Width of the reference image in pixels *)
		nRefImageHeight	:	UDINT;	(* Height of the reference image in pixels *)
		ipEdgePoints	:	REFERENCE TO ITcVnContainer;	(* Returns a container with the 4 edge points of the reference image transformed into the coordinates of the source image (ContainerType_Vector_TcVnPoint2_REAL) *)
		fMaxDist	:	REAL;	(* Maximum allowed descriptor distance (-1 disables this filter criterion) *)
		fMaxKnnRatio	:	REAL;	(* Maximum allowed distance ratio between first and second best match ([0..1], -1 disables this filter criterion) *)
		eNormType	:	ETcVnNormalizationType;	(* Normalization type used for descriptor matching (HAMMING recommended for AKAZE, ORB, and BRISK. HAMMING2 is recommended for ORB if the ORB nBriefPoints parameter is 3 or 4. ) *)
		eAlgorithm	:	ETcVnEstimationAlgorithm;	(* Estimation algorithm used for computing the perspective transformation between the two point sets *)
		fReprojThreshold	:	LREAL;	(* Maximum allowed reprojection error to treat a point pair as an inlier (only used if eAlgorithm is RANSAC, RHO) *)
		nMaxIterations	:	UDINT;	(* Maximum number of RANSAC iterations *)
		fConfidence	:	LREAL;	(* Confidence (0..1) *)
		ipGoodMatches	:	REFERENCE TO ITcVnContainer;	(* Returns a container with good matches (optional, set to 0 if not required; ContainerType_Vector_TcVnDMatch) *)
		ipInlierMask	:	REFERENCE TO ITcVnContainer;	(* Returns a mask marking the inliers (optional, set to 0 if not required; ContainerType_Vector_SINT; only for RANSAC, LMEDS) *)
		hrPrev	:	HRESULT;	(* HRESULT indicating the result of previous operations (If SUCCEEDED(hrPrev) equals false, no operation is executed.) *)
	END_VAR
	VAR_OUTPUT
		aPerspectiveTransform	:	TcVnMatrix3x3_LREAL;	(* Returns the perspective transformation matrix, which transforms the reference points to the source points  *)
		nNumberOfGoodMatches	:	UDINT;	(* Return the number of good matches *)
		nNumberOfInliers	:	UDINT;	(* Return the number of inlier matches *)
	END_VAR

END_FUNCTION

// Functions/Keypoint Features/F_VN_FindReferenceKeyPointsInImageAKAZE

	{attribute 'TcIecLibraryType'}
	{attribute 'external_name' := 'F_VN_FindReferenceKeyPointsInImageAKAZE_GUID_3E60BF9E_414B_2D4A_590B_404373E8C146'}
	(* Searches a reference image, represented by its AKAZE keypoints and corresponding descriptors, in a given source image (uses the default TcVnParamsAKAZE parameters). *)
	FUNCTION F_VN_FindReferenceKeyPointsInImageAKAZE : HRESULT
	VAR_INPUT
		ipSrcImage	:	ITcVnImage;	(* Source image *)
		ipRefKeyPoints	:	ITcVnContainer;	(* KeyPoints of the reference image, e.g. computed with F_VN_KeyPointsAndDescriptorsAKAZE (ContainerType_Vector_TcVnKeyPoint) *)
		ipRefDescriptors	:	ITcVnImage;	(* Descriptors of the reference image KeyPoints, e.g. computed with F_VN_KeyPointsAndDescriptorsAKAZE *)
		nRefImageWidth	:	UDINT;	(* Width of the reference image in pixels *)
		nRefImageHeight	:	UDINT;	(* Height of the reference image in pixels *)
		ipEdgePoints	:	REFERENCE TO ITcVnContainer;	(* Returns a container with the 4 edge points of the reference image transformed into ipSrcImage coordinates (ContainerType_Vector_TcVnPoint2_REAL) *)
		fMaxDist	:	REAL;	(* Maximum allowed descriptor distance (-1 disables this filter criterion) *)
		fMaxKnnRatio	:	REAL;	(* Maximum allowed distance ratio between first and second best match ([0..1], -1 disables this filter criterion) *)
		hrPrev	:	HRESULT;	(* HRESULT indicating the result of previous operations (If SUCCEEDED(hrPrev) equals false, no operation is executed.) *)
	END_VAR
	VAR_OUTPUT
		aPerspectiveTransform	:	TcVnMatrix3x3_LREAL;	(* Returns the perspective transformation matrix, which transforms the reference points to the source points *)
		nNumberOfGoodMatches	:	UDINT;	(* Return the number of good matches *)
		nNumberOfInliers	:	UDINT;	(* Return the number of inlier matches *)
	END_VAR

END_FUNCTION

// Functions/Keypoint Features/F_VN_KeyPointsAndDescriptorsAKAZE

	{attribute 'TcIecLibraryType'}
	{attribute 'external_name' := 'F_VN_KeyPointsAndDescriptorsAKAZE_GUID_B41C4895_6ADD_2EB5_67E5_9C8930AEEECE'}
	(* Detects keypoints and compute descriptors using the AKAZE method. *)
	FUNCTION F_VN_KeyPointsAndDescriptorsAKAZE : HRESULT
	VAR_INPUT
		ipSrcImage	:	ITcVnImage;	(* Source image *)
		ipKeyPoints	:	REFERENCE TO ITcVnContainer;	(* Returns a container which is filled with the keypoints (ContainerType_Vector_TcVnKeyPoint; Non-zero interface pointers are reused.) *)
		ipDescriptors	:	REFERENCE TO ITcVnImage;	(* Descriptor image (set to 0 if not required; 1 descriptor in each row; An appropriate image will be created if required.) *)
		hrPrev	:	HRESULT;	(* HRESULT indicating the result of previous operations (If SUCCEEDED(hrPrev) equals false, no operation is executed.) *)
	END_VAR

END_FUNCTION

// Functions/Keypoint Features/F_VN_FindReferenceKeyPointsInImageAKAZEExp

	{attribute 'TcIecLibraryType'}
	{attribute 'external_name' := 'F_VN_FindReferenceKeyPointsInImageAKAZEExp_GUID_DDC005BA_01EC_2612_4CC4_D1D09E600488'}
	(* Searches a reference image, represented by its AKAZE keypoints and corresponding descriptors, in a given source image. (expert function) *)
	FUNCTION F_VN_FindReferenceKeyPointsInImageAKAZEExp : HRESULT
	VAR_INPUT
		ipSrcImage	:	ITcVnImage;	(* Source image *)
		ipRefKeyPoints	:	ITcVnContainer;	(* KeyPoints of the reference image, e.g. computed with F_VN_KeyPointsAndDescriptorsAKAZE (ContainerType_Vector_TcVnKeyPoint) *)
		ipRefDescriptors	:	ITcVnImage;	(* Descriptors of the reference image KeyPoints, e.g. computed with F_VN_KeyPointsAndDescriptorsAKAZE *)
		nRefImageWidth	:	UDINT;	(* Width of the reference image in pixels *)
		nRefImageHeight	:	UDINT;	(* Height of the reference image in pixels *)
		ipEdgePoints	:	REFERENCE TO ITcVnContainer;	(* Returns a container with the 4 edge points of the reference image transformed into ipSrcImage coordinates (ContainerType_Vector_TcVnPoint2_REAL) *)
		fMaxDist	:	REAL;	(* Maximum allowed descriptor distance (-1 disables this filter criterion) *)
		fMaxKnnRatio	:	REAL;	(* Maximum allowed distance ratio between first and second best match ([0..1], -1 disables this filter criterion) *)
		eNormType	:	ETcVnNormalizationType;	(* Normalization type used for descriptor matching *)
		ipSrcImageMask	:	ITcVnImage;	(* Mask to specify, where to look for keypoints in ipSrcImage (set to 0 if no mask required) *)
	END_VAR
	VAR_IN_OUT
		stAkazeParams	:	TcVnParamsAKAZE;	(* Parameters to configure the keypoint and descriptor computation for ipSrcImage (resulting descriptors must be compatible to ipRefDescriptors!) *)
	END_VAR
	VAR_INPUT
		eAlgorithm	:	ETcVnEstimationAlgorithm;	(* Estimation algorithm used for computing the perspective transformation between the two point sets *)
		fReprojThreshold	:	LREAL;	(* Maximum allowed reprojection error to treat a point pair as an inlier (only used if eAlgorithm is RANSAC, RHO) *)
		nMaxIterations	:	UDINT;	(* Maximum number of RANSAC iterations *)
		fConfidence	:	LREAL;	(* Confidence (0..1) *)
		hrPrev	:	HRESULT;	(* HRESULT indicating the result of previous operations (If SUCCEEDED(hrPrev) equals false, no operation is executed.) *)
	END_VAR
	VAR_OUTPUT
		aPerspectiveTransform	:	TcVnMatrix3x3_LREAL;	(* Returns the perspective transformation matrix, which transforms the reference points to the source points  *)
		nNumberOfGoodMatches	:	UDINT;	(* Return the number of good matches *)
		nNumberOfInliers	:	UDINT;	(* Return the number of inlier matches *)
	END_VAR

END_FUNCTION

// Functions/Keypoint Features/F_VN_FindReferenceKeyPointsInImageBRISK

	{attribute 'TcIecLibraryType'}
	{attribute 'external_name' := 'F_VN_FindReferenceKeyPointsInImageBRISK_GUID_4154D295_530F_22BF_66B9_DF803FAC4482'}
	(* Searches a reference image, represented by its BRISK keypoints and corresponding descriptors, in a given source image (uses the default TcVnParamsBRISK parameters). *)
	FUNCTION F_VN_FindReferenceKeyPointsInImageBRISK : HRESULT
	VAR_INPUT
		ipSrcImage	:	ITcVnImage;	(* Source image *)
		ipRefKeyPoints	:	ITcVnContainer;	(* KeyPoints of the reference image, e.g. computed with F_VN_KeyPointsAndDescriptorsBRISK (ContainerType_Vector_TcVnKeyPoint) *)
		ipRefDescriptors	:	ITcVnImage;	(* Descriptors of the reference image KeyPoints, e.g. computed with F_VN_KeyPointsAndDescriptorsBRISK *)
		nRefImageWidth	:	UDINT;	(* Width of the reference image in pixels *)
		nRefImageHeight	:	UDINT;	(* Height of the reference image in pixels *)
		ipEdgePoints	:	REFERENCE TO ITcVnContainer;	(* Returns a container with the 4 edge points of the reference image transformed into ipSrcImage coordinates (ContainerType_Vector_TcVnPoint2_REAL) *)
		fMaxDist	:	REAL;	(* Maximum allowed descriptor distance (-1 disables this filter criterion) *)
		fMaxKnnRatio	:	REAL;	(* Maximum allowed distance ratio between first and second best match ([0..1], -1 disables this filter criterion) *)
		hrPrev	:	HRESULT;	(* HRESULT indicating the result of previous operations (If SUCCEEDED(hrPrev) equals false, no operation is executed.) *)
	END_VAR
	VAR_OUTPUT
		aPerspectiveTransform	:	TcVnMatrix3x3_LREAL;	(* Returns the perspective transformation matrix, which transforms the reference points to the source points  *)
		nNumberOfGoodMatches	:	UDINT;	(* Return the number of good matches *)
		nNumberOfInliers	:	UDINT;	(* Return the number of inlier matches *)
	END_VAR

END_FUNCTION

// Functions/Keypoint Features/F_VN_KeyPointsAndDescriptorsBRISK

	{attribute 'TcIecLibraryType'}
	{attribute 'external_name' := 'F_VN_KeyPointsAndDescriptorsBRISK_GUID_03200E19_CF13_28E7_57F0_1FD556F83DCE'}
	(* Detects keypoints and compute descriptors using the BRISK method. *)
	FUNCTION F_VN_KeyPointsAndDescriptorsBRISK : HRESULT
	VAR_INPUT
		ipSrcImage	:	ITcVnImage;	(* Source image *)
		ipKeyPoints	:	REFERENCE TO ITcVnContainer;	(* Returns a container which is filled with the keypoints (ContainerType_Vector_TcVnKeyPoint; Non-zero interface pointers are reused.) *)
		ipDescriptors	:	REFERENCE TO ITcVnImage;	(* Descriptor image (set to 0 if not required; 1 descriptor in each row; An appropriate image will be created if required.) *)
		hrPrev	:	HRESULT;	(* HRESULT indicating the result of previous operations (If SUCCEEDED(hrPrev) equals false, no operation is executed.) *)
	END_VAR

END_FUNCTION

// Functions/Keypoint Features/F_VN_FindReferenceKeyPointsInImageBRISKExp

	{attribute 'TcIecLibraryType'}
	{attribute 'external_name' := 'F_VN_FindReferenceKeyPointsInImageBRISKExp_GUID_03587FF7_1B71_2663_4B6D_F4CF1BD375D1'}
	(* Searches a reference image, represented by its BRISK keypoints and corresponding descriptors, in a given source image. (expert function) *)
	FUNCTION F_VN_FindReferenceKeyPointsInImageBRISKExp : HRESULT
	VAR_INPUT
		ipSrcImage	:	ITcVnImage;	(* Source image *)
		ipRefKeyPoints	:	ITcVnContainer;	(* KeyPoints of the reference image, e.g. computed with F_VN_KeyPointsAndDescriptorsBRISK (ContainerType_Vector_TcVnKeyPoint) *)
		ipRefDescriptors	:	ITcVnImage;	(* Descriptors of the reference image KeyPoints, e.g. computed with F_VN_KeyPointsAndDescriptorsBRISK *)
		nRefImageWidth	:	UDINT;	(* Width of the reference image in pixels *)
		nRefImageHeight	:	UDINT;	(* Height of the reference image in pixels *)
		ipEdgePoints	:	REFERENCE TO ITcVnContainer;	(* Returns a container with the 4 edge points of the reference image transformed into ipSrcImage coordinates (ContainerType_Vector_TcVnPoint2_REAL) *)
		fMaxDist	:	REAL;	(* Maximum allowed descriptor distance (-1 disables this filter criterion) *)
		fMaxKnnRatio	:	REAL;	(* Maximum allowed distance ratio between first and second best match ([0..1], -1 disables this filter criterion) *)
		eNormType	:	ETcVnNormalizationType;	(* Normalization type used for descriptor matching *)
		ipSrcImageMask	:	ITcVnImage;	(* Mask to specify, where to look for keypoints in ipSrcImage (set to 0 if no mask required) *)
	END_VAR
	VAR_IN_OUT
		stBriskParams	:	TcVnParamsBRISK;	(* Parameters to configure the keypoint and descriptor computation for ipSrcImage (resulting descriptors must be compatible to ipRefDescriptors!) *)
	END_VAR
	VAR_INPUT
		eAlgorithm	:	ETcVnEstimationAlgorithm;	(* Estimation algorithm used for computing the perspective transformation between the two point sets *)
		fReprojThreshold	:	LREAL;	(* Maximum allowed reprojection error to treat a point pair as an inlier (only used if eAlgorithm is RANSAC, RHO) *)
		nMaxIterations	:	UDINT;	(* Maximum number of RANSAC iterations *)
		fConfidence	:	LREAL;	(* Confidence (0..1) *)
		hrPrev	:	HRESULT;	(* HRESULT indicating the result of previous operations (If SUCCEEDED(hrPrev) equals false, no operation is executed.) *)
	END_VAR
	VAR_OUTPUT
		aPerspectiveTransform	:	TcVnMatrix3x3_LREAL;	(* Returns the perspective transformation matrix, which transforms the reference points to the source points  *)
		nNumberOfGoodMatches	:	UDINT;	(* Return the number of good matches *)
		nNumberOfInliers	:	UDINT;	(* Return the number of inlier matches *)
	END_VAR

END_FUNCTION

// Functions/Keypoint Features/F_VN_FindReferenceKeyPointsInImageORB

	{attribute 'TcIecLibraryType'}
	{attribute 'external_name' := 'F_VN_FindReferenceKeyPointsInImageORB_GUID_20150D05_604A_2C01_618C_CFE9911A223E'}
	(* Searches a reference image, represented by its ORB keypoints and corresponding descriptors, in a given source image (uses the default TcVnParamsORB parameters). *)
	FUNCTION F_VN_FindReferenceKeyPointsInImageORB : HRESULT
	VAR_INPUT
		ipSrcImage	:	ITcVnImage;	(* Source image *)
		ipRefKeyPoints	:	ITcVnContainer;	(* KeyPoints of the reference image, e.g. computed with F_VN_KeyPointsAndDescriptorsORB (ContainerType_Vector_TcVnKeyPoint) *)
		ipRefDescriptors	:	ITcVnImage;	(* Descriptors of the reference image KeyPoints, e.g. computed with F_VN_KeyPointsAndDescriptorsORB *)
		nRefImageWidth	:	UDINT;	(* Width of the reference image in pixels *)
		nRefImageHeight	:	UDINT;	(* Height of the reference image in pixels *)
		ipEdgePoints	:	REFERENCE TO ITcVnContainer;	(* Returns a container with the 4 edge points of the reference image transformed into ipSrcImage coordinates (ContainerType_Vector_TcVnPoint2_REAL) *)
		fMaxDist	:	REAL;	(* Maximum allowed descriptor distance (-1 disables this filter criterion) *)
		fMaxKnnRatio	:	REAL;	(* Maximum allowed distance ratio between first and second best match ([0..1], -1 disables this filter criterion) *)
		hrPrev	:	HRESULT;	(* HRESULT indicating the result of previous operations (If SUCCEEDED(hrPrev) equals false, no operation is executed.) *)
	END_VAR
	VAR_OUTPUT
		aPerspectiveTransform	:	TcVnMatrix3x3_LREAL;	(* Returns the perspective transformation matrix, which transforms the reference points to the source points  *)
		nNumberOfGoodMatches	:	UDINT;	(* Return the number of good matches *)
		nNumberOfInliers	:	UDINT;	(* Return the number of inlier matches *)
	END_VAR

END_FUNCTION

// Functions/Keypoint Features/F_VN_KeyPointsAndDescriptorsORB

	{attribute 'TcIecLibraryType'}
	{attribute 'external_name' := 'F_VN_KeyPointsAndDescriptorsORB_GUID_18B65A24_0127_2980_57E2_3D87371ABE16'}
	(* Detects keypoints and compute descriptors using the ORB method. *)
	FUNCTION F_VN_KeyPointsAndDescriptorsORB : HRESULT
	VAR_INPUT
		ipSrcImage	:	ITcVnImage;	(* Source image *)
		ipKeyPoints	:	REFERENCE TO ITcVnContainer;	(* Returns a container which is filled with the keypoints (ContainerType_Vector_TcVnKeyPoint; Non-zero interface pointers are reused.) *)
		ipDescriptors	:	REFERENCE TO ITcVnImage;	(* Descriptor image (set to 0 if not required; 1 descriptor in each row; An appropriate image will be created if required.) *)
		hrPrev	:	HRESULT;	(* HRESULT indicating the result of previous operations (If SUCCEEDED(hrPrev) equals false, no operation is executed.) *)
	END_VAR

END_FUNCTION

// Functions/Keypoint Features/F_VN_FindReferenceKeyPointsInImageORBExp

	{attribute 'TcIecLibraryType'}
	{attribute 'external_name' := 'F_VN_FindReferenceKeyPointsInImageORBExp_GUID_FD11A86C_3A56_2660_6227_D3F82C7EA5DF'}
	(* Searches a reference image, represented by its ORB keypoints and corresponding descriptors, in a given source image. (expert function) *)
	FUNCTION F_VN_FindReferenceKeyPointsInImageORBExp : HRESULT
	VAR_INPUT
		ipSrcImage	:	ITcVnImage;	(* Source image *)
		ipRefKeyPoints	:	ITcVnContainer;	(* KeyPoints of the reference image, e.g. computed with F_VN_KeyPointsAndDescriptorsORB (ContainerType_Vector_TcVnKeyPoint) *)
		ipRefDescriptors	:	ITcVnImage;	(* Descriptors of the reference image KeyPoints, e.g. computed with F_VN_KeyPointsAndDescriptorsORB *)
		nRefImageWidth	:	UDINT;	(* Width of the reference image in pixels *)
		nRefImageHeight	:	UDINT;	(* Height of the reference image in pixels *)
		ipEdgePoints	:	REFERENCE TO ITcVnContainer;	(* Returns a container with the 4 edge points of the reference image transformed into ipSrcImage coordinates (ContainerType_Vector_TcVnPoint2_REAL) *)
		fMaxDist	:	REAL;	(* Maximum allowed descriptor distance (-1 disables this filter criterion) *)
		fMaxKnnRatio	:	REAL;	(* Maximum allowed distance ratio between first and second best match ([0..1], -1 disables this filter criterion) *)
		eNormType	:	ETcVnNormalizationType;	(* Normalization type used for descriptor matching (HAMMING recommended for ORB, HAMMING2 if the ORB nBriefPoints parameter is 3 or 4) *)
		ipSrcImageMask	:	ITcVnImage;	(* Mask to specify, where to look for keypoints in ipSrcImage (set to 0 if no mask required) *)
	END_VAR
	VAR_IN_OUT
		stOrbParams	:	TcVnParamsORB;	(* Parameters to configure the keypoint and descriptor computation for ipSrcImage (resulting descriptors must be compatible to ipRefDescriptors!) *)
	END_VAR
	VAR_INPUT
		eAlgorithm	:	ETcVnEstimationAlgorithm;	(* Estimation algorithm used for computing the perspective transformation between the two point sets *)
		fReprojThreshold	:	LREAL;	(* Maximum allowed reprojection error to treat a point pair as an inlier (only used if eAlgorithm is RANSAC, RHO) *)
		nMaxIterations	:	UDINT;	(* Maximum number of RANSAC iterations *)
		fConfidence	:	LREAL;	(* Confidence (0..1) *)
		hrPrev	:	HRESULT;	(* HRESULT indicating the result of previous operations (If SUCCEEDED(hrPrev) equals false, no operation is executed.) *)
	END_VAR
	VAR_OUTPUT
		aPerspectiveTransform	:	TcVnMatrix3x3_LREAL;	(* Returns the perspective transformation matrix, which transforms the reference points to the source points  *)
		nNumberOfGoodMatches	:	UDINT;	(* Return the number of good matches *)
		nNumberOfInliers	:	UDINT;	(* Return the number of inlier matches *)
	END_VAR

END_FUNCTION

// Functions/Keypoint Features/F_VN_GetMatchCoordinates

	{attribute 'TcIecLibraryType'}
	{attribute 'external_name' := 'F_VN_GetMatchCoordinates_GUID_4F6CA593_3230_214D_6D56_D5E7B477B525'}
	(* Return the coordinates of keypoints that match each other. *)
	FUNCTION F_VN_GetMatchCoordinates : HRESULT
	VAR_INPUT
		ipQueryKeyPoints	:	ITcVnContainer;	(* Container with query Keypoints (i.e. keypoints of a reference/template image) of type CTcVnContainer_Vector_TcVnKeyPoint *)
		ipTrainKeyPoints	:	ITcVnContainer;	(* Container with training Keypoints (i.e. keypoints of a source/input image) of type CTcVnContainer_Vector_TcVnKeyPoint *)
		ipMatches	:	ITcVnContainer;	(* Container with matches between query and train Keypoints (CTcVnContainer_Vector_TcVnDMatch). *)
		ipQueryCoordinates	:	REFERENCE TO ITcVnContainer;	(* Returns a container with the coordinates of keypoints from the query Keypoints that exist in ipMatches (CTcVnContainer_Vector_TcVnPoint2_REAL) *)
		ipTrainCoordinates	:	REFERENCE TO ITcVnContainer;	(* Returns a container with the coordinates of keypoints from the training Keypoints that exist in ipMatches (CTcVnContainer_Vector_TcVnPoint2_REAL) *)
		hrPrev	:	HRESULT;	(* HRESULT indicating the result of previous operations (If SUCCEEDED(hrPrev) equals false, no operation is executed.) *)
	END_VAR

END_FUNCTION

// Functions/Keypoint Features/F_VN_KeyPointsAGAST

	{attribute 'TcIecLibraryType'}
	{attribute 'external_name' := 'F_VN_KeyPointsAGAST_GUID_0CFD7A2D_1288_2D8F_56FE_768C07F02FFC'}
	(* Detects keypoints using the AGAST method. *)
	FUNCTION F_VN_KeyPointsAGAST : HRESULT
	VAR_INPUT
		ipSrcImage	:	ITcVnImage;	(* Source image *)
		ipKeyPoints	:	REFERENCE TO ITcVnContainer;	(* Returns a container which is filled with the keypoints (ContainerType_Vector_TcVnKeyPoint; Non-zero interface pointers are reused.) *)
		hrPrev	:	HRESULT;	(* HRESULT indicating the result of previous operations (If SUCCEEDED(hrPrev) equals false, no operation is executed.) *)
	END_VAR

END_FUNCTION

// Functions/Keypoint Features/F_VN_KeyPointsAGASTExp

	{attribute 'TcIecLibraryType'}
	{attribute 'external_name' := 'F_VN_KeyPointsAGASTExp_GUID_1B873B00_9D41_2BA4_6CC1_FB15F3CA8B93'}
	(* Detects keypoints using the AGAST method. (expert function) *)
	FUNCTION F_VN_KeyPointsAGASTExp : HRESULT
	VAR_INPUT
		ipSrcImage	:	ITcVnImage;	(* Source image *)
		ipKeyPoints	:	REFERENCE TO ITcVnContainer;	(* Returns a container which is filled with the keypoints (ContainerType_Vector_TcVnKeyPoint; Non-zero interface pointers are reused.) *)
		ipMask	:	ITcVnImage;	(* Mask to specify, where to look for keypoints (set to 0 if no mask required) *)
	END_VAR
	VAR_IN_OUT
		stParams	:	TcVnParamsAGAST;	(* Additional expert parameters *)
	END_VAR
	VAR_INPUT
		hrPrev	:	HRESULT;	(* HRESULT indicating the result of previous operations (If SUCCEEDED(hrPrev) equals false, no operation is executed.) *)
	END_VAR

END_FUNCTION

// Functions/Keypoint Features/F_VN_KeyPointsAndDescriptorsAKAZEExp

	{attribute 'TcIecLibraryType'}
	{attribute 'external_name' := 'F_VN_KeyPointsAndDescriptorsAKAZEExp_GUID_EC168E6D_1EBE_24E6_5B61_F6A2ED5AA1C2'}
	(* Detects keypoints and compute descriptors using the AKAZE method. (expert function) *)
	FUNCTION F_VN_KeyPointsAndDescriptorsAKAZEExp : HRESULT
	VAR_INPUT
		ipSrcImage	:	ITcVnImage;	(* Source image *)
		ipKeyPoints	:	REFERENCE TO ITcVnContainer;	(* Returns a container which is filled with the keypoints (ContainerType_Vector_TcVnKeyPoint; Non-zero interface pointers are reused.) *)
		ipDescriptors	:	REFERENCE TO ITcVnImage;	(* Descriptor image (set to 0 if not required; 1 descriptor in each row; An appropriate image will be created if required.) *)
		ipMask	:	ITcVnImage;	(* Mask to specify, where to look for keypoints (set to 0 if no mask required) *)
	END_VAR
	VAR_IN_OUT
		stParams	:	TcVnParamsAKAZE;	(* Additional expert parameters *)
	END_VAR
	VAR_INPUT
		hrPrev	:	HRESULT;	(* HRESULT indicating the result of previous operations (If SUCCEEDED(hrPrev) equals false, no operation is executed.) *)
	END_VAR

END_FUNCTION

// Functions/Keypoint Features/F_VN_KeyPointsAndDescriptorsBRISKExp

	{attribute 'TcIecLibraryType'}
	{attribute 'external_name' := 'F_VN_KeyPointsAndDescriptorsBRISKExp_GUID_5D8D7ED8_AD2E_2F1A_799F_F6057C98614E'}
	(* Detects keypoints and compute descriptors using the BRISK method. (expert function) *)
	FUNCTION F_VN_KeyPointsAndDescriptorsBRISKExp : HRESULT
	VAR_INPUT
		ipSrcImage	:	ITcVnImage;	(* Source image *)
		ipKeyPoints	:	REFERENCE TO ITcVnContainer;	(* Returns a container which is filled with the keypoints (ContainerType_Vector_TcVnKeyPoint; Non-zero interface pointers are reused.) *)
		ipDescriptors	:	REFERENCE TO ITcVnImage;	(* Descriptor image (set to 0 if not required; 1 descriptor in each row; An appropriate image will be created if required.) *)
		ipMask	:	ITcVnImage;	(* Mask to specify, where to look for keypoints (set to 0 if no mask required) *)
	END_VAR
	VAR_IN_OUT
		stParams	:	TcVnParamsBRISK;	(* Additional expert parameters *)
	END_VAR
	VAR_INPUT
		hrPrev	:	HRESULT;	(* HRESULT indicating the result of previous operations (If SUCCEEDED(hrPrev) equals false, no operation is executed.) *)
	END_VAR

END_FUNCTION

// Functions/Keypoint Features/F_VN_KeyPointsAndDescriptorsKAZE

